  [248] = {x=67.075, y=92.051, z=16.707, rx=-170.912, ry=12.532, rz=153, fatherId=fPrdFrame[0]}
  [249] = {x=69.882, y=92.045, z=17.386, rx=-170.899, ry=12.987, rz=153, fatherId=fPrdFrame[0]}
  [250] = {x=72.688, y=92.04, z=18.091, rx=-170.885, ry=13.443, rz=153, fatherId=fPrdFrame[0]}
  [251] = {x=75.494, y=92.033, z=18.821, rx=-170.871, ry=13.9, rz=153, fatherId=fPrdFrame[0]}
  [252] = {x=78.301, y=92.027, z=19.576, rx=-170.856, ry=14.358, rz=153, fatherId=fPrdFrame[0]}
  [253] = {x=81.107, y=92.021, z=20.356, rx=-170.841, ry=14.816, rz=153, fatherId=fPrdFrame[0]}
  [254] = {x=83.913, y=92.014, z=21.163, rx=-170.825, ry=15.276, rz=153, fatherId=fPrdFrame[0]}
  [255] = {x=86.72, y=92.007, z=21.995, rx=-170.809, ry=15.737, rz=153, fatherId=fPrdFrame[0]}
  [256] = {x=89.526, y=91.999, z=22.854, rx=-170.792, ry=16.198, rz=153, fatherId=fPrdFrame[0]}
  [257] = {x=92.332, y=91.992, z=23.738, rx=-170.774, ry=16.661, rz=153, fatherId=fPrdFrame[0]}
  [258] = {x=95.139, y=91.984, z=24.649, rx=-170.756, ry=17.125, rz=153, fatherId=fPrdFrame[0]}
  [259] = {x=97.945, y=91.976, z=25.587, rx=-170.737, ry=17.59, rz=153, fatherId=fPrdFrame[0]}
  [260] = {x=97.937, y=94.85, z=26.084, rx=-170.445, ry=17.608, rz=153, fatherId=fPrdFrame[0]}
  [261] = {x=95.131, y=94.859, z=25.145, rx=-170.465, ry=17.142, rz=153, fatherId=fPrdFrame[0]}
  [262] = {x=92.325, y=94.867, z=24.233, rx=-170.483, ry=16.678, rz=153, fatherId=fPrdFrame[0]}
  [263] = {x=89.519, y=94.874, z=23.348, rx=-170.501, ry=16.215, rz=153, fatherId=fPrdFrame[0]}
  [264] = {x=86.713, y=94.882, z=22.488, rx=-170.519, ry=15.753, rz=153, fatherId=fPrdFrame[0]}
  [265] = {x=83.907, y=94.889, z=21.655, rx=-170.536, ry=15.292, rz=153, fatherId=fPrdFrame[0]}
  [266] = {x=81.101, y=94.896, z=20.848, rx=-170.552, ry=14.831, rz=153, fatherId=fPrdFrame[0]}
  [267] = {x=78.294, y=94.903, z=20.066, rx=-170.568, ry=14.372, rz=153, fatherId=fPrdFrame[0]}
  [268] = {x=75.488, y=94.909, z=19.31, rx=-170.583, ry=13.914, rz=153, fatherId=fPrdFrame[0]}
  [269] = {x=72.682, y=94.916, z=18.58, rx=-170.598, ry=13.457, rz=153, fatherId=fPrdFrame[0]}
  [270] = {x=69.876, y=94.922, z=17.875, rx=-170.612, ry=13, rz=153, fatherId=fPrdFrame[0]}
  [271] = {x=67.07, y=94.928, z=17.195, rx=-170.625, ry=12.545, rz=153, fatherId=fPrdFrame[0]}
  [272] = {x=64.264, y=94.933, z=16.54, rx=-170.638, ry=12.09, rz=153, fatherId=fPrdFrame[0]}
  [273] = {x=61.458, y=94.939, z=15.909, rx=-170.65, ry=11.636, rz=153, fatherId=fPrdFrame[0]}
  [274] = {x=58.652, y=94.944, z=15.304, rx=-170.662, ry=11.182, rz=153, fatherId=fPrdFrame[0]}
  [275] = {x=55.846, y=94.949, z=14.723, rx=-170.674, ry=10.73, rz=153, fatherId=fPrdFrame[0]}
  [276] = {x=53.04, y=94.953, z=14.167, rx=-170.685, ry=10.278, rz=153, fatherId=fPrdFrame[0]}
  [277] = {x=50.233, y=94.958, z=13.635, rx=-170.695, ry=9.826, rz=153, fatherId=fPrdFrame[0]}
  [278] = {x=47.427, y=94.962, z=13.128, rx=-170.705, ry=9.376, rz=153, fatherId=fPrdFrame[0]}
  [279] = {x=44.621, y=94.966, z=12.645, rx=-170.714, ry=8.925, rz=153, fatherId=fPrdFrame[0]}
  [280] = {x=41.815, y=94.97, z=12.185, rx=-170.723, ry=8.476, rz=153, fatherId=fPrdFrame[0]}
  [281] = {x=39.009, y=94.974, z=11.75, rx=-170.732, ry=8.027, rz=153, fatherId=fPrdFrame[0]}
  [282] = {x=36.203, y=94.977, z=11.339, rx=-170.74, ry=7.578, rz=153, fatherId=fPrdFrame[0]}
  [283] = {x=33.397, y=94.98, z=10.952, rx=-170.747, ry=7.13, rz=153, fatherId=fPrdFrame[0]}
  [284] = {x=30.591, y=94.983, z=10.589, rx=-170.754, ry=6.682, rz=153, fatherId=fPrdFrame[0]}
  [285] = {x=27.785, y=94.986, z=10.249, rx=-170.761, ry=6.235, rz=153, fatherId=fPrdFrame[0]}
  [286] = {x=24.979, y=94.989, z=9.933, rx=-170.767, ry=5.788, rz=153, fatherId=fPrdFrame[0]}
  [287] = {x=22.173, y=94.991, z=9.641, rx=-170.772, ry=5.342, rz=153, fatherId=fPrdFrame[0]}
  [288] = {x=19.367, y=94.993, z=9.372, rx=-170.777, ry=4.895, rz=153, fatherId=fPrdFrame[0]}
  [289] = {x=16.561, y=94.995, z=9.127, rx=-170.782, ry=4.449, rz=153, fatherId=fPrdFrame[0]}
  [290] = {x=13.755, y=94.997, z=8.905, rx=-170.786, ry=4.004, rz=153, fatherId=fPrdFrame[0]}
  [291] = {x=10.948, y=94.999, z=8.707, rx=-170.79, ry=3.558, rz=153, fatherId=fPrdFrame[0]}
  [292] = {x=8.142, y=95, z=8.532, rx=-170.793, ry=3.113, rz=153, fatherId=fPrdFrame[0]}
  [293] = {x=5.336, y=95.001, z=8.381, rx=-170.796, ry=2.668, rz=153, fatherId=fPrdFrame[0]}
  [294] = {x=2.53, y=95.002, z=8.253, rx=-170.799, ry=2.223, rz=153, fatherId=fPrdFrame[0]}
  [295] = {x=-0.276, y=95.003, z=8.148, rx=-170.801, ry=1.778, rz=153, fatherId=fPrdFrame[0]}
  [296] = {x=-3.082, y=95.004, z=8.066, rx=-170.802, ry=1.334, rz=153, fatherId=fPrdFrame[0]}
  [297] = {x=-5.888, y=95.004, z=8.008, rx=-170.803, ry=0.889, rz=153, fatherId=fPrdFrame[0]}
  [298] = {x=-8.694, y=95.005, z=7.973, rx=-170.804, ry=0.444, rz=153, fatherId=fPrdFrame[0]}
  [299] = {x=-11.5, y=95.005, z=7.962, rx=-170.804, rz=153, fatherId=fPrdFrame[0]}
  [300] = {x=-14.306, y=95.005, z=7.973, rx=-170.804, ry=-0.444, rz=153, fatherId=fPrdFrame[0]}
  [301] = {x=-17.112, y=95.004, z=8.008, rx=-170.803, ry=-0.889, rz=153, fatherId=fPrdFrame[0]}
  [302] = {x=-19.918, y=95.004, z=8.066, rx=-170.802, ry=-1.334, rz=153, fatherId=fPrdFrame[0]}
  [303] = {x=-22.724, y=95.003, z=8.148, rx=-170.801, ry=-1.778, rz=153, fatherId=fPrdFrame[0]}
  [304] = {x=-25.53, y=95.002, z=8.253, rx=-170.799, ry=-2.223, rz=153, fatherId=fPrdFrame[0]}
  [305] = {x=-28.336, y=95.001, z=8.381, rx=-170.796, ry=-2.668, rz=153, fatherId=fPrdFrame[0]}
  [306] = {x=-31.142, y=95, z=8.532, rx=-170.793, ry=-3.113, rz=153, fatherId=fPrdFrame[0]}
  [307] = {x=-33.948, y=94.999, z=8.707, rx=-170.79, ry=-3.558, rz=153, fatherId=fPrdFrame[0]}
  [308] = {x=-36.755, y=94.997, z=8.905, rx=-170.786, ry=-4.004, rz=153, fatherId=fPrdFrame[0]}
  [309] = {x=-39.561, y=94.995, z=9.127, rx=-170.782, ry=-4.449, rz=153, fatherId=fPrdFrame[0]}
  [310] = {x=-42.367, y=94.993, z=9.372, rx=-170.777, ry=-4.895, rz=153, fatherId=fPrdFrame[0]}
  [311] = {x=-45.173, y=94.991, z=9.641, rx=-170.772, ry=-5.342, rz=153, fatherId=fPrdFrame[0]}
  [312] = {x=-47.979, y=94.989, z=9.933, rx=-170.767, ry=-5.788, rz=153, fatherId=fPrdFrame[0]}
  [313] = {x=-50.785, y=94.986, z=10.249, rx=-170.761, ry=-6.235, rz=153, fatherId=fPrdFrame[0]}
  [314] = {x=-53.591, y=94.983, z=10.589, rx=-170.754, ry=-6.682, rz=153, fatherId=fPrdFrame[0]}
  [315] = {x=-56.397, y=94.98, z=10.952, rx=-170.747, ry=-7.13, rz=153, fatherId=fPrdFrame[0]}
  [316] = {x=-59.203, y=94.977, z=11.339, rx=-170.74, ry=-7.578, rz=153, fatherId=fPrdFrame[0]}
  [317] = {x=-62.009, y=94.974, z=11.75, rx=-170.732, ry=-8.027, rz=153, fatherId=fPrdFrame[0]}
  [318] = {x=-64.815, y=94.97, z=12.185, rx=-170.723, ry=-8.476, rz=153, fatherId=fPrdFrame[0]}
  [319] = {x=-67.621, y=94.966, z=12.645, rx=-170.714, ry=-8.925, rz=153, fatherId=fPrdFrame[0]}
  [320] = {x=-70.427, y=94.962, z=13.128, rx=-170.705, ry=-9.376, rz=153, fatherId=fPrdFrame[0]}
  [321] = {x=-73.233, y=94.958, z=13.635, rx=-170.695, ry=-9.826, rz=153, fatherId=fPrdFrame[0]}
  [322] = {x=-76.04, y=94.953, z=14.167, rx=-170.685, ry=-10.278, rz=153, fatherId=fPrdFrame[0]}
  [323] = {x=-78.846, y=94.949, z=14.723, rx=-170.674, ry=-10.73, rz=153, fatherId=fPrdFrame[0]}
  [324] = {x=-81.652, y=94.944, z=15.304, rx=-170.662, ry=-11.182, rz=153, fatherId=fPrdFrame[0]}
  [325] = {x=-84.458, y=94.939, z=15.909, rx=-170.65, ry=-11.636, rz=153, fatherId=fPrdFrame[0]}
  [326] = {x=-87.264, y=94.933, z=16.54, rx=-170.638, ry=-12.09, rz=153, fatherId=fPrdFrame[0]}
  [327] = {x=-90.07, y=94.928, z=17.195, rx=-170.625, ry=-12.545, rz=153, fatherId=fPrdFrame[0]}
  [328] = {x=-92.876, y=94.922, z=17.875, rx=-170.612, ry=-13, rz=153, fatherId=fPrdFrame[0]}
  [329] = {x=-95.682, y=94.916, z=18.58, rx=-170.598, ry=-13.457, rz=153, fatherId=fPrdFrame[0]}
  [330] = {x=-98.488, y=94.909, z=19.31, rx=-170.583, ry=-13.914, rz=153, fatherId=fPrdFrame[0]}
  [331] = {x=-101.294, y=94.903, z=20.066, rx=-170.568, ry=-14.372, rz=153, fatherId=fPrdFrame[0]}
  [332] = {x=-104.101, y=94.896, z=20.848, rx=-170.552, ry=-14.831, rz=153, fatherId=fPrdFrame[0]}
  [333] = {x=-106.907, y=94.889, z=21.655, rx=-170.536, ry=-15.292, rz=153, fatherId=fPrdFrame[0]}
  [334] = {x=-109.713, y=94.882, z=22.488, rx=-170.519, ry=-15.753, rz=153, fatherId=fPrdFrame[0]}
  [335] = {x=-112.519, y=94.874, z=23.348, rx=-170.501, ry=-16.215, rz=153, fatherId=fPrdFrame[0]}
  [336] = {x=-115.325, y=94.867, z=24.233, rx=-170.483, ry=-16.678, rz=153, fatherId=fPrdFrame[0]}
  [337] = {x=-118.131, y=94.859, z=25.145, rx=-170.465, ry=-17.142, rz=153, fatherId=fPrdFrame[0]}
  [338] = {x=-120.937, y=94.85, z=26.084, rx=-170.445, ry=-17.608, rz=153, fatherId=fPrdFrame[0]}
  [339] = {x=-120.93, y=97.724, z=26.597, rx=-170.153, ry=-17.627, rz=153, fatherId=fPrdFrame[0]}
  [340] = {x=-118.124, y=97.733, z=25.657, rx=-170.173, ry=-17.161, rz=153, fatherId=fPrdFrame[0]}
  [341] = {x=-115.318, y=97.741, z=24.744, rx=-170.192, ry=-16.696, rz=153, fatherId=fPrdFrame[0]}
  [342] = {x=-112.512, y=97.749, z=23.857, rx=-170.211, ry=-16.232, rz=153, fatherId=fPrdFrame[0]}
  [343] = {x=-109.706, y=97.757, z=22.997, rx=-170.229, ry=-15.769, rz=153, fatherId=fPrdFrame[0]}
  [344] = {x=-106.9, y=97.765, z=22.163, rx=-170.246, ry=-15.308, rz=153, fatherId=fPrdFrame[0]}
  [345] = {x=-104.094, y=97.772, z=21.355, rx=-170.263, ry=-14.847, rz=153, fatherId=fPrdFrame[0]}
  [346] = {x=-101.288, y=97.779, z=20.572, rx=-170.279, ry=-14.387, rz=153, fatherId=fPrdFrame[0]}
  [347] = {x=-98.482, y=97.786, z=19.816, rx=-170.295, ry=-13.929, rz=153, fatherId=fPrdFrame[0]}
  [348] = {x=-95.676, y=97.792, z=19.084, rx=-170.31, ry=-13.471, rz=153, fatherId=fPrdFrame[0]}
  [349] = {x=-92.87, y=97.798, z=18.378, rx=-170.324, ry=-13.014, rz=153, fatherId=fPrdFrame[0]}
  [350] = {x=-90.064, y=97.804, z=17.698, rx=-170.338, ry=-12.558, rz=153, fatherId=fPrdFrame[0]}
  [351] = {x=-87.259, y=97.81, z=17.042, rx=-170.352, ry=-12.102, rz=153, fatherId=fPrdFrame[0]}
  [352] = {x=-84.453, y=97.815, z=16.411, rx=-170.364, ry=-11.648, rz=153, fatherId=fPrdFrame[0]}
  [353] = {x=-81.647, y=97.821, z=15.805, rx=-170.377, ry=-11.194, rz=153, fatherId=fPrdFrame[0]}
  [354] = {x=-78.841, y=97.826, z=15.224, rx=-170.389, ry=-10.741, rz=153, fatherId=fPrdFrame[0]}
  [355] = {x=-76.035, y=97.831, z=14.667, rx=-170.4, ry=-10.288, rz=153, fatherId=fPrdFrame[0]}
  [356] = {x=-73.229, y=97.835, z=14.134, rx=-170.41, ry=-9.837, rz=153, fatherId=fPrdFrame[0]}
  [357] = {x=-70.423, y=97.84, z=13.626, rx=-170.421, ry=-9.385, rz=153, fatherId=fPrdFrame[0]}
  [358] = {x=-67.617, y=97.844, z=13.143, rx=-170.43, ry=-8.935, rz=153, fatherId=fPrdFrame[0]}
  [359] = {x=-64.811, y=97.848, z=12.683, rx=-170.44, ry=-8.485, rz=153, fatherId=fPrdFrame[0]}
  [360] = {x=-62.005, y=97.852, z=12.248, rx=-170.448, ry=-8.035, rz=153, fatherId=fPrdFrame[0]}
  [361] = {x=-59.2, y=97.855, z=11.836, rx=-170.456, ry=-7.586, rz=153, fatherId=fPrdFrame[0]}
  [362] = {x=-56.394, y=97.858, z=11.448, rx=-170.464, ry=-7.137, rz=153, fatherId=fPrdFrame[0]}
  [363] = {x=-53.588, y=97.861, z=11.085, rx=-170.471, ry=-6.689, rz=153, fatherId=fPrdFrame[0]}
  [364] = {x=-50.782, y=97.864, z=10.745, rx=-170.478, ry=-6.242, rz=153, fatherId=fPrdFrame[0]}
  [365] = {x=-47.976, y=97.867, z=10.428, rx=-170.484, ry=-5.794, rz=153, fatherId=fPrdFrame[0]}
  [366] = {x=-45.17, y=97.87, z=10.136, rx=-170.49, ry=-5.347, rz=153, fatherId=fPrdFrame[0]}
  [367] = {x=-42.364, y=97.872, z=9.867, rx=-170.495, ry=-4.9, rz=153, fatherId=fPrdFrame[0]}
  [368] = {x=-39.559, y=97.874, z=9.621, rx=-170.5, ry=-4.454, rz=153, fatherId=fPrdFrame[0]}
  [369] = {x=-36.753, y=97.876, z=9.399, rx=-170.505, ry=-4.008, rz=153, fatherId=fPrdFrame[0]}
  [370] = {x=-33.947, y=97.877, z=9.201, rx=-170.509, ry=-3.562, rz=153, fatherId=fPrdFrame[0]}
  [371] = {x=-31.141, y=97.879, z=9.026, rx=-170.512, ry=-3.116, rz=153, fatherId=fPrdFrame[0]}
  [372] = {x=-28.335, y=97.88, z=8.874, rx=-170.515, ry=-2.671, rz=153, fatherId=fPrdFrame[0]}
  [373] = {x=-25.529, y=97.881, z=8.746, rx=-170.517, ry=-2.225, rz=153, fatherId=fPrdFrame[0]}
  [374] = {x=-22.723, y=97.882, z=8.641, rx=-170.52, ry=-1.78, rz=153, fatherId=fPrdFrame[0]}
  [375] = {x=-19.918, y=97.883, z=8.56, rx=-170.521, ry=-1.335, rz=153, fatherId=fPrdFrame[0]}
  [376] = {x=-17.112, y=97.883, z=8.501, rx=-170.522, ry=-0.89, rz=153, fatherId=fPrdFrame[0]}
  [377] = {x=-14.306, y=97.884, z=8.466, rx=-170.523, ry=-0.445, rz=153, fatherId=fPrdFrame[0]}
  [378] = {x=-11.5, y=97.884, z=8.455, rx=-170.523, rz=153, fatherId=fPrdFrame[0]}
  [379] = {x=-8.694, y=97.884, z=8.466, rx=-170.523, ry=0.445, rz=153, fatherId=fPrdFrame[0]}
  [380] = {x=-5.888, y=97.883, z=8.501, rx=-170.522, ry=0.89, rz=153, fatherId=fPrdFrame[0]}
  [381] = {x=-3.082, y=97.883, z=8.56, rx=-170.521, ry=1.335, rz=153, fatherId=fPrdFrame[0]}
  [382] = {x=-0.277, y=97.882, z=8.641, rx=-170.52, ry=1.78, rz=153, fatherId=fPrdFrame[0]}
  [383] = {x=2.529, y=97.881, z=8.746, rx=-170.517, ry=2.225, rz=153, fatherId=fPrdFrame[0]}
  [384] = {x=5.335, y=97.88, z=8.874, rx=-170.515, ry=2.671, rz=153, fatherId=fPrdFrame[0]}
  [385] = {x=8.141, y=97.879, z=9.026, rx=-170.512, ry=3.116, rz=153, fatherId=fPrdFrame[0]}
  [386] = {x=10.947, y=97.877, z=9.201, rx=-170.509, ry=3.562, rz=153, fatherId=fPrdFrame[0]}
  [387] = {x=13.753, y=97.876, z=9.399, rx=-170.505, ry=4.008, rz=153, fatherId=fPrdFrame[0]}
  [388] = {x=16.559, y=97.874, z=9.621, rx=-170.5, ry=4.454, rz=153, fatherId=fPrdFrame[0]}
  [389] = {x=19.364, y=97.872, z=9.867, rx=-170.495, ry=4.9, rz=153, fatherId=fPrdFrame[0]}
  [390] = {x=22.17, y=97.87, z=10.136, rx=-170.49, ry=5.347, rz=153, fatherId=fPrdFrame[0]}
  [391] = {x=24.976, y=97.867, z=10.428, rx=-170.484, ry=5.794, rz=153, fatherId=fPrdFrame[0]}
  [392] = {x=27.782, y=97.864, z=10.745, rx=-170.478, ry=6.242, rz=153, fatherId=fPrdFrame[0]}
  [393] = {x=30.588, y=97.861, z=11.085, rx=-170.471, ry=6.689, rz=153, fatherId=fPrdFrame[0]}
  [394] = {x=33.394, y=97.858, z=11.448, rx=-170.464, ry=7.137, rz=153, fatherId=fPrdFrame[0]}
  [395] = {x=36.2, y=97.855, z=11.836, rx=-170.456, ry=7.586, rz=153, fatherId=fPrdFrame[0]}
  [396] = {x=39.005, y=97.852, z=12.248, rx=-170.448, ry=8.035, rz=153, fatherId=fPrdFrame[0]}
  [397] = {x=41.811, y=97.848, z=12.683, rx=-170.44, ry=8.485, rz=153, fatherId=fPrdFrame[0]}
  [398] = {x=44.617, y=97.844, z=13.143, rx=-170.43, ry=8.935, rz=153, fatherId=fPrdFrame[0]}
  [399] = {x=47.423, y=97.84, z=13.626, rx=-170.421, ry=9.385, rz=153, fatherId=fPrdFrame[0]}
  [400] = {x=50.229, y=97.835, z=14.134, rx=-170.41, ry=9.837, rz=153, fatherId=fPrdFrame[0]}
  [401] = {x=53.035, y=97.831, z=14.667, rx=-170.4, ry=10.288, rz=153, fatherId=fPrdFrame[0]}
  [402] = {x=55.841, y=97.826, z=15.224, rx=-170.389, ry=10.741, rz=153, fatherId=fPrdFrame[0]}
  [403] = {x=58.647, y=97.821, z=15.805, rx=-170.377, ry=11.194, rz=153, fatherId=fPrdFrame[0]}
  [404] = {x=61.453, y=97.815, z=16.411, rx=-170.364, ry=11.648, rz=153, fatherId=fPrdFrame[0]}
  [405] = {x=64.259, y=97.81, z=17.042, rx=-170.352, ry=12.102, rz=153, fatherId=fPrdFrame[0]}
  [406] = {x=67.064, y=97.804, z=17.698, rx=-170.338, ry=12.558, rz=153, fatherId=fPrdFrame[0]}
  [407] = {x=69.87, y=97.798, z=18.378, rx=-170.324, ry=13.014, rz=153, fatherId=fPrdFrame[0]}
  [408] = {x=72.676, y=97.792, z=19.084, rx=-170.31, ry=13.471, rz=153, fatherId=fPrdFrame[0]}
  [409] = {x=75.482, y=97.786, z=19.816, rx=-170.295, ry=13.929, rz=153, fatherId=fPrdFrame[0]}
  [410] = {x=78.288, y=97.779, z=20.572, rx=-170.279, ry=14.387, rz=153, fatherId=fPrdFrame[0]}
  [411] = {x=81.094, y=97.772, z=21.355, rx=-170.263, ry=14.847, rz=153, fatherId=fPrdFrame[0]}
  [412] = {x=83.9, y=97.765, z=22.163, rx=-170.246, ry=15.308, rz=153, fatherId=fPrdFrame[0]}
  [413] = {x=86.706, y=97.757, z=22.997, rx=-170.229, ry=15.769, rz=153, fatherId=fPrdFrame[0]}
  [414] = {x=89.512, y=97.749, z=23.857, rx=-170.211, ry=16.232, rz=153, fatherId=fPrdFrame[0]}
  [415] = {x=92.318, y=97.741, z=24.744, rx=-170.192, ry=16.696, rz=153, fatherId=fPrdFrame[0]}
  [416] = {x=95.124, y=97.733, z=25.657, rx=-170.173, ry=17.161, rz=153, fatherId=fPrdFrame[0]}
  [417] = {x=97.93, y=97.724, z=26.597, rx=-170.153, ry=17.627, rz=153, fatherId=fPrdFrame[0]}
  [418] = {x=97.922, y=100.599, z=27.126, rx=-169.86, ry=17.646, rz=153, fatherId=fPrdFrame[0]}
  [419] = {x=95.116, y=100.607, z=26.185, rx=-169.881, ry=17.179, rz=153, fatherId=fPrdFrame[0]}
  [420] = {x=92.31, y=100.616, z=25.271, rx=-169.9, ry=16.714, rz=153, fatherId=fPrdFrame[0]}
  [421] = {x=89.504, y=100.624, z=24.383, rx=-169.92, ry=16.25, rz=153, fatherId=fPrdFrame[0]}
  [422] = {x=86.699, y=100.632, z=23.522, rx=-169.938, ry=15.786, rz=153, fatherId=fPrdFrame[0]}
  [423] = {x=83.893, y=100.64, z=22.687, rx=-169.956, ry=15.324, rz=153, fatherId=fPrdFrame[0]}
  [424] = {x=81.087, y=100.647, z=21.877, rx=-169.974, ry=14.863, rz=153, fatherId=fPrdFrame[0]}
  [425] = {x=78.281, y=100.655, z=21.094, rx=-169.99, ry=14.403, rz=153, fatherId=fPrdFrame[0]}
  [426] = {x=75.476, y=100.662, z=20.337, rx=-170.006, ry=13.944, rz=153, fatherId=fPrdFrame[0]}
  [427] = {x=72.67, y=100.668, z=19.604, rx=-170.022, ry=13.485, rz=153, fatherId=fPrdFrame[0]}
  [428] = {x=69.864, y=100.675, z=18.898, rx=-170.037, ry=13.028, rz=153, fatherId=fPrdFrame[0]}
  [429] = {x=67.059, y=100.681, z=18.216, rx=-170.051, ry=12.571, rz=153, fatherId=fPrdFrame[0]}
  [430] = {x=64.253, y=100.687, z=17.56, rx=-170.065, ry=12.116, rz=153, fatherId=fPrdFrame[0]}
  [431] = {x=61.447, y=100.692, z=16.928, rx=-170.078, ry=11.66, rz=153, fatherId=fPrdFrame[0]}
  [432] = {x=58.642, y=100.698, z=16.321, rx=-170.091, ry=11.206, rz=153, fatherId=fPrdFrame[0]}
  [433] = {x=55.836, y=100.703, z=15.739, rx=-170.103, ry=10.752, rz=153, fatherId=fPrdFrame[0]}
  [434] = {x=53.03, y=100.708, z=15.182, rx=-170.115, ry=10.3, rz=153, fatherId=fPrdFrame[0]}
  [435] = {x=50.224, y=100.713, z=14.649, rx=-170.126, ry=9.847, rz=153, fatherId=fPrdFrame[0]}
  [436] = {x=47.419, y=100.717, z=14.14, rx=-170.136, ry=9.396, rz=153, fatherId=fPrdFrame[0]}
  [437] = {x=44.613, y=100.722, z=13.656, rx=-170.146, ry=8.944, rz=153, fatherId=fPrdFrame[0]}
  [438] = {x=41.807, y=100.726, z=13.196, rx=-170.156, ry=8.494, rz=153, fatherId=fPrdFrame[0]}
  [439] = {x=39.002, y=100.73, z=12.76, rx=-170.165, ry=8.044, rz=153, fatherId=fPrdFrame[0]}
  [440] = {x=36.196, y=100.733, z=12.348, rx=-170.173, ry=7.594, rz=153, fatherId=fPrdFrame[0]}
  [441] = {x=33.39, y=100.737, z=11.96, rx=-170.181, ry=7.145, rz=153, fatherId=fPrdFrame[0]}
  [442] = {x=30.585, y=100.74, z=11.596, rx=-170.188, ry=6.696, rz=153, fatherId=fPrdFrame[0]}
  [443] = {x=27.779, y=100.743, z=11.256, rx=-170.195, ry=6.248, rz=153, fatherId=fPrdFrame[0]}
  [444] = {x=24.973, y=100.746, z=10.939, rx=-170.202, ry=5.8, rz=153, fatherId=fPrdFrame[0]}
  [445] = {x=22.168, y=100.748, z=10.646, rx=-170.208, ry=5.353, rz=153, fatherId=fPrdFrame[0]}
  [446] = {x=19.362, y=100.75, z=10.377, rx=-170.213, ry=4.906, rz=153, fatherId=fPrdFrame[0]}
  [447] = {x=16.556, y=100.753, z=10.131, rx=-170.218, ry=4.459, rz=153, fatherId=fPrdFrame[0]}
  [448] = {x=13.751, y=100.754, z=9.909, rx=-170.223, ry=4.012, rz=153, fatherId=fPrdFrame[0]}
  [449] = {x=10.945, y=100.756, z=9.71, rx=-170.227, ry=3.566, rz=153, fatherId=fPrdFrame[0]}
  [450] = {x=8.14, y=100.758, z=9.535, rx=-170.23, ry=3.12, rz=153, fatherId=fPrdFrame[0]}
  [451] = {x=5.334, y=100.759, z=9.383, rx=-170.233, ry=2.674, rz=153, fatherId=fPrdFrame[0]}
  [452] = {x=2.528, y=100.76, z=9.255, rx=-170.236, ry=2.228, rz=153, fatherId=fPrdFrame[0]}
  [453] = {x=-0.277, y=100.761, z=9.15, rx=-170.238, ry=1.782, rz=153, fatherId=fPrdFrame[0]}
  [454] = {x=-3.083, y=100.762, z=9.068, rx=-170.24, ry=1.336, rz=153, fatherId=fPrdFrame[0]}
  [455] = {x=-5.889, y=100.762, z=9.01, rx=-170.241, ry=0.891, rz=153, fatherId=fPrdFrame[0]}
  [456] = {x=-8.694, y=100.763, z=8.975, rx=-170.242, ry=0.445, rz=153, fatherId=fPrdFrame[0]}
  [457] = {x=-11.5, y=100.763, z=8.963, rx=-170.242, rz=153, fatherId=fPrdFrame[0]}
  [458] = {x=-14.306, y=100.763, z=8.975, rx=-170.242, ry=-0.445, rz=153, fatherId=fPrdFrame[0]}
  [459] = {x=-17.111, y=100.762, z=9.01, rx=-170.241, ry=-0.891, rz=153, fatherId=fPrdFrame[0]}
  [460] = {x=-19.917, y=100.762, z=9.068, rx=-170.24, ry=-1.336, rz=153, fatherId=fPrdFrame[0]}
  [461] = {x=-22.723, y=100.761, z=9.15, rx=-170.238, ry=-1.782, rz=153, fatherId=fPrdFrame[0]}
  [462] = {x=-25.528, y=100.76, z=9.255, rx=-170.236, ry=-2.228, rz=153, fatherId=fPrdFrame[0]}
  [463] = {x=-28.334, y=100.759, z=9.383, rx=-170.233, ry=-2.674, rz=153, fatherId=fPrdFrame[0]}
  [464] = {x=-31.14, y=100.758, z=9.535, rx=-170.23, ry=-3.12, rz=153, fatherId=fPrdFrame[0]}
  [465] = {x=-33.945, y=100.756, z=9.71, rx=-170.227, ry=-3.566, rz=153, fatherId=fPrdFrame[0]}
  [466] = {x=-36.751, y=100.754, z=9.909, rx=-170.223, ry=-4.012, rz=153, fatherId=fPrdFrame[0]}
  [467] = {x=-39.556, y=100.753, z=10.131, rx=-170.218, ry=-4.459, rz=153, fatherId=fPrdFrame[0]}
  [468] = {x=-42.362, y=100.75, z=10.377, rx=-170.213, ry=-4.906, rz=153, fatherId=fPrdFrame[0]}
  [469] = {x=-45.168, y=100.748, z=10.646, rx=-170.208, ry=-5.353, rz=153, fatherId=fPrdFrame[0]}
  [470] = {x=-47.973, y=100.746, z=10.939, rx=-170.202, ry=-5.8, rz=153, fatherId=fPrdFrame[0]}
  [471] = {x=-50.779, y=100.743, z=11.256, rx=-170.195, ry=-6.248, rz=153, fatherId=fPrdFrame[0]}
  [472] = {x=-53.585, y=100.74, z=11.596, rx=-170.188, ry=-6.696, rz=153, fatherId=fPrdFrame[0]}
  [473] = {x=-56.39, y=100.737, z=11.96, rx=-170.181, ry=-7.145, rz=153, fatherId=fPrdFrame[0]}
  [474] = {x=-59.196, y=100.733, z=12.348, rx=-170.173, ry=-7.594, rz=153, fatherId=fPrdFrame[0]}
  [475] = {x=-62.002, y=100.73, z=12.76, rx=-170.165, ry=-8.044, rz=153, fatherId=fPrdFrame[0]}
  [476] = {x=-64.807, y=100.726, z=13.196, rx=-170.156, ry=-8.494, rz=153, fatherId=fPrdFrame[0]}
  [477] = {x=-67.613, y=100.722, z=13.656, rx=-170.146, ry=-8.944, rz=153, fatherId=fPrdFrame[0]}
  [478] = {x=-70.419, y=100.717, z=14.14, rx=-170.136, ry=-9.396, rz=153, fatherId=fPrdFrame[0]}
  [479] = {x=-73.224, y=100.713, z=14.649, rx=-170.126, ry=-9.847, rz=153, fatherId=fPrdFrame[0]}
  [480] = {x=-76.03, y=100.708, z=15.182, rx=-170.115, ry=-10.3, rz=153, fatherId=fPrdFrame[0]}
  [481] = {x=-78.836, y=100.703, z=15.739, rx=-170.103, ry=-10.752, rz=153, fatherId=fPrdFrame[0]}
  [482] = {x=-81.642, y=100.698, z=16.321, rx=-170.091, ry=-11.206, rz=153, fatherId=fPrdFrame[0]}
  [483] = {x=-84.447, y=100.692, z=16.928, rx=-170.078, ry=-11.66, rz=153, fatherId=fPrdFrame[0]}
  [484] = {x=-87.253, y=100.687, z=17.56, rx=-170.065, ry=-12.116, rz=153, fatherId=fPrdFrame[0]}
  [485] = {x=-90.059, y=100.681, z=18.216, rx=-170.051, ry=-12.571, rz=153, fatherId=fPrdFrame[0]}
  [486] = {x=-92.864, y=100.675, z=18.898, rx=-170.037, ry=-13.028, rz=153, fatherId=fPrdFrame[0]}
  [487] = {x=-95.67, y=100.668, z=19.604, rx=-170.022, ry=-13.485, rz=153, fatherId=fPrdFrame[0]}
  [488] = {x=-98.476, y=100.662, z=20.337, rx=-170.006, ry=-13.944, rz=153, fatherId=fPrdFrame[0]}
  [489] = {x=-101.281, y=100.655, z=21.094, rx=-169.99, ry=-14.403, rz=153, fatherId=fPrdFrame[0]}
  [490] = {x=-104.087, y=100.647, z=21.877, rx=-169.974, ry=-14.863, rz=153, fatherId=fPrdFrame[0]}
  [491] = {x=-106.893, y=100.64, z=22.687, rx=-169.956, ry=-15.324, rz=153, fatherId=fPrdFrame[0]}
  [492] = {x=-109.699, y=100.632, z=23.522, rx=-169.938, ry=-15.786, rz=153, fatherId=fPrdFrame[0]}
  [493] = {x=-112.504, y=100.624, z=24.383, rx=-169.92, ry=-16.25, rz=153, fatherId=fPrdFrame[0]}
  [494] = {x=-115.31, y=100.616, z=25.271, rx=-169.9, ry=-16.714, rz=153, fatherId=fPrdFrame[0]}
  [495] = {x=-118.116, y=100.607, z=26.185, rx=-169.881, ry=-17.179, rz=153, fatherId=fPrdFrame[0]}
  [496] = {x=-120.922, y=100.599, z=27.126, rx=-169.86, ry=-17.646, rz=153, fatherId=fPrdFrame[0]}
  [497] = {x=-120.922, y=100.599, z=77.126, rx=-169.86, ry=-17.646, rz=153, fatherId=fPrdFrame[0]}
  [498] = {x=19.385, y=66.207, z=5.253, rx=-173.587, ry=4.853, rz=153, fatherId=fPrdFrame[0]}
  [499] = {x=16.577, y=66.209, z=5.01, rx=-173.59, ry=4.411, rz=153, fatherId=fPrdFrame[0]}
  [500] = {x=13.769, y=66.21, z=4.79, rx=-173.593, ry=3.969, rz=153, fatherId=fPrdFrame[0]}
  [501] = {x=10.962, y=66.211, z=4.594, rx=-173.595, ry=3.528, rz=153, fatherId=fPrdFrame[0]}
  [502] = {x=8.154, y=66.212, z=4.42, rx=-173.598, ry=3.086, rz=153, fatherId=fPrdFrame[0]}
  [503] = {x=5.346, y=66.213, z=4.27, rx=-173.6, ry=2.645, rz=153, fatherId=fPrdFrame[0]}
  [504] = {x=2.539, y=66.214, z=4.143, rx=-173.601, ry=2.204, rz=153, fatherId=fPrdFrame[0]}
  [505] = {x=-0.269, y=66.214, z=4.039, rx=-173.603, ry=1.763, rz=153, fatherId=fPrdFrame[0]}
  [506] = {x=-3.077, y=66.215, z=3.958, rx=-173.604, ry=1.322, rz=153, fatherId=fPrdFrame[0]}
  [507] = {x=-5.885, y=66.215, z=3.901, rx=-173.605, ry=0.881, rz=153, fatherId=fPrdFrame[0]}
  [508] = {x=-8.692, y=66.215, z=3.866, rx=-173.605, ry=0.441, rz=153, fatherId=fPrdFrame[0]}
  [509] = {x=-11.5, y=66.215, z=3.855, rx=-173.605, rz=153, fatherId=fPrdFrame[0]}
  [510] = {x=-14.308, y=66.215, z=3.866, rx=-173.605, ry=-0.441, rz=153, fatherId=fPrdFrame[0]}
  [511] = {x=-17.115, y=66.215, z=3.901, rx=-173.605, ry=-0.881, rz=153, fatherId=fPrdFrame[0]}
  [512] = {x=-19.923, y=66.215, z=3.958, rx=-173.604, ry=-1.322, rz=153, fatherId=fPrdFrame[0]}
  [513] = {x=-22.731, y=66.214, z=4.039, rx=-173.603, ry=-1.763, rz=153, fatherId=fPrdFrame[0]}
  [514] = {x=-25.539, y=66.214, z=4.143, rx=-173.601, ry=-2.204, rz=153, fatherId=fPrdFrame[0]}
  [515] = {x=-28.346, y=66.213, z=4.27, rx=-173.6, ry=-2.645, rz=153, fatherId=fPrdFrame[0]}
  [516] = {x=-31.154, y=66.212, z=4.42, rx=-173.598, ry=-3.086, rz=153, fatherId=fPrdFrame[0]}
  [517] = {x=-33.962, y=66.211, z=4.594, rx=-173.595, ry=-3.528, rz=153, fatherId=fPrdFrame[0]}
  [518] = {x=-36.769, y=66.21, z=4.79, rx=-173.593, ry=-3.969, rz=153, fatherId=fPrdFrame[0]}
  [519] = {x=-39.577, y=66.209, z=5.01, rx=-173.59, ry=-4.411, rz=153, fatherId=fPrdFrame[0]}
  [520] = {x=-42.385, y=66.207, z=5.253, rx=-173.587, ry=-4.853, rz=153, fatherId=fPrdFrame[0]}
  [521] = {x=-45.193, y=66.206, z=5.519, rx=-173.583, ry=-5.296, rz=153, fatherId=fPrdFrame[0]}
  [522] = {x=-48, y=66.204, z=5.809, rx=-173.579, ry=-5.738, rz=153, fatherId=fPrdFrame[0]}
  [523] = {x=-50.808, y=66.202, z=6.122, rx=-173.575, ry=-6.181, rz=153, fatherId=fPrdFrame[0]}
  [524] = {x=-53.616, y=66.2, z=6.459, rx=-173.57, ry=-6.625, rz=153, fatherId=fPrdFrame[0]}
  [525] = {x=-56.424, y=66.198, z=6.819, rx=-173.566, ry=-7.069, rz=153, fatherId=fPrdFrame[0]}
  [526] = {x=-59.231, y=66.196, z=7.203, rx=-173.56, ry=-7.513, rz=153, fatherId=fPrdFrame[0]}
  [527] = {x=-62.039, y=66.194, z=7.611, rx=-173.555, ry=-7.958, rz=153, fatherId=fPrdFrame[0]}
  [528] = {x=-64.847, y=66.191, z=8.042, rx=-173.549, ry=-8.403, rz=153, fatherId=fPrdFrame[0]}
  [529] = {x=-67.654, y=66.189, z=8.497, rx=-173.543, ry=-8.848, rz=153, fatherId=fPrdFrame[0]}
  [530] = {x=-70.462, y=66.186, z=8.976, rx=-173.536, ry=-9.295, rz=153, fatherId=fPrdFrame[0]}
  [531] = {x=-73.27, y=66.183, z=9.479, rx=-173.53, ry=-9.742, rz=153, fatherId=fPrdFrame[0]}
  [532] = {x=-76.078, y=66.18, z=10.006, rx=-173.522, ry=-10.189, rz=153, fatherId=fPrdFrame[0]}
  [533] = {x=-78.885, y=66.176, z=10.557, rx=-173.515, ry=-10.637, rz=153, fatherId=fPrdFrame[0]}
  [534] = {x=-81.693, y=66.173, z=11.133, rx=-173.507, ry=-11.086, rz=153, fatherId=fPrdFrame[0]}
  [535] = {x=-84.501, y=66.169, z=11.733, rx=-173.499, ry=-11.535, rz=153, fatherId=fPrdFrame[0]}
  [536] = {x=-87.309, y=66.166, z=12.358, rx=-173.49, ry=-11.985, rz=153, fatherId=fPrdFrame[0]}
  [537] = {x=-90.116, y=66.162, z=13.007, rx=-173.481, ry=-12.436, rz=153, fatherId=fPrdFrame[0]}
  [538] = {x=-92.924, y=66.158, z=13.681, rx=-173.472, ry=-12.887, rz=153, fatherId=fPrdFrame[0]}
  [539] = {x=-95.732, y=66.154, z=14.38, rx=-173.462, ry=-13.34, rz=153, fatherId=fPrdFrame[0]}
  [540] = {x=-98.54, y=66.149, z=15.103, rx=-173.452, ry=-13.793, rz=153, fatherId=fPrdFrame[0]}
  [541] = {x=-101.347, y=66.145, z=15.853, rx=-173.442, ry=-14.247, rz=153, fatherId=fPrdFrame[0]}
  [542] = {x=-104.155, y=66.14, z=16.627, rx=-173.431, ry=-14.702, rz=153, fatherId=fPrdFrame[0]}
  [543] = {x=-106.963, y=66.135, z=17.427, rx=-173.419, ry=-15.158, rz=153, fatherId=fPrdFrame[0]}
  [544] = {x=-109.771, y=66.13, z=18.253, rx=-173.408, ry=-15.615, rz=153, fatherId=fPrdFrame[0]}
  [545] = {x=-112.578, y=66.125, z=19.104, rx=-173.396, ry=-16.073, rz=153, fatherId=fPrdFrame[0]}
  [546] = {x=-115.386, y=66.119, z=19.981, rx=-173.383, ry=-16.532, rz=153, fatherId=fPrdFrame[0]}
  [547] = {x=-118.194, y=66.114, z=20.885, rx=-173.37, ry=-16.992, rz=153, fatherId=fPrdFrame[0]}
  [548] = {x=-121.002, y=66.108, z=21.815, rx=-173.357, ry=-17.454, rz=153, fatherId=fPrdFrame[0]}
  [549] = {x=-120.996, y=68.982, z=22.172, rx=-173.067, ry=-17.466, rz=153, fatherId=fPrdFrame[0]}
  [550] = {x=-118.189, y=68.988, z=21.241, rx=-173.081, ry=-17.005, rz=153, fatherId=fPrdFrame[0]}
  [551] = {x=-115.381, y=68.994, z=20.337, rx=-173.094, ry=-16.544, rz=153, fatherId=fPrdFrame[0]}
  [552] = {x=-112.573, y=69, z=19.459, rx=-173.107, ry=-16.085, rz=153, fatherId=fPrdFrame[0]}
  [553] = {x=-109.766, y=69.005, z=18.607, rx=-173.12, ry=-15.627, rz=153, fatherId=fPrdFrame[0]}
  [554] = {x=-106.958, y=69.01, z=17.781, rx=-173.132, ry=-15.169, rz=153, fatherId=fPrdFrame[0]}
  [555] = {x=-104.151, y=69.016, z=16.98, rx=-173.144, ry=-14.713, rz=153, fatherId=fPrdFrame[0]}
  [556] = {x=-101.343, y=69.02, z=16.205, rx=-173.155, ry=-14.258, rz=153, fatherId=fPrdFrame[0]}
  [557] = {x=-98.535, y=69.025, z=15.455, rx=-173.166, ry=-13.803, rz=153, fatherId=fPrdFrame[0]}
  [558] = {x=-95.728, y=69.03, z=14.731, rx=-173.177, ry=-13.35, rz=153, fatherId=fPrdFrame[0]}
  [559] = {x=-92.92, y=69.034, z=14.032, rx=-173.187, ry=-12.897, rz=153, fatherId=fPrdFrame[0]}
  [560] = {x=-90.112, y=69.038, z=13.357, rx=-173.196, ry=-12.445, rz=153, fatherId=fPrdFrame[0]}
  [561] = {x=-87.305, y=69.042, z=12.707, rx=-173.206, ry=-11.994, rz=153, fatherId=fPrdFrame[0]}
  [562] = {x=-84.497, y=69.046, z=12.082, rx=-173.215, ry=-11.543, rz=153, fatherId=fPrdFrame[0]}
  [563] = {x=-81.69, y=69.05, z=11.482, rx=-173.223, ry=-11.094, rz=153, fatherId=fPrdFrame[0]}
  [564] = {x=-78.882, y=69.054, z=10.906, rx=-173.232, ry=-10.645, rz=153, fatherId=fPrdFrame[0]}
  [565] = {x=-76.074, y=69.057, z=10.354, rx=-173.239, ry=-10.196, rz=153, fatherId=fPrdFrame[0]}
  [566] = {x=-73.267, y=69.06, z=9.827, rx=-173.247, ry=-9.749, rz=153, fatherId=fPrdFrame[0]}
  [567] = {x=-70.459, y=69.063, z=9.323, rx=-173.254, ry=-9.301, rz=153, fatherId=fPrdFrame[0]}
  [568] = {x=-67.652, y=69.066, z=8.844, rx=-173.261, ry=-8.855, rz=153, fatherId=fPrdFrame[0]}
  [569] = {x=-64.844, y=69.069, z=8.389, rx=-173.267, ry=-8.409, rz=153, fatherId=fPrdFrame[0]}
  [570] = {x=-62.037, y=69.072, z=7.957, rx=-173.273, ry=-7.963, rz=153, fatherId=fPrdFrame[0]}
  [571] = {x=-59.229, y=69.074, z=7.549, rx=-173.279, ry=-7.518, rz=153, fatherId=fPrdFrame[0]}
  [572] = {x=-56.421, y=69.077, z=7.165, rx=-173.285, ry=-7.074, rz=153, fatherId=fPrdFrame[0]}
  [573] = {x=-53.614, y=69.079, z=6.805, rx=-173.29, ry=-6.63, rz=153, fatherId=fPrdFrame[0]}
  [574] = {x=-50.806, y=69.081, z=6.468, rx=-173.294, ry=-6.186, rz=153, fatherId=fPrdFrame[0]}
  [575] = {x=-47.999, y=69.083, z=6.154, rx=-173.299, ry=-5.742, rz=153, fatherId=fPrdFrame[0]}
  [576] = {x=-45.191, y=69.084, z=5.864, rx=-173.303, ry=-5.299, rz=153, fatherId=fPrdFrame[0]}
  [577] = {x=-42.383, y=69.086, z=5.598, rx=-173.306, ry=-4.857, rz=153, fatherId=fPrdFrame[0]}
  [578] = {x=-39.576, y=69.087, z=5.354, rx=-173.31, ry=-4.414, rz=153, fatherId=fPrdFrame[0]}
  [579] = {x=-36.768, y=69.089, z=5.135, rx=-173.313, ry=-3.972, rz=153, fatherId=fPrdFrame[0]}
  [580] = {x=-33.961, y=69.09, z=4.938, rx=-173.316, ry=-3.53, rz=153, fatherId=fPrdFrame[0]}
  [581] = {x=-31.153, y=69.091, z=4.764, rx=-173.318, ry=-3.088, rz=153, fatherId=fPrdFrame[0]}
  [582] = {x=-28.345, y=69.092, z=4.614, rx=-173.32, ry=-2.647, rz=153, fatherId=fPrdFrame[0]}
  [583] = {x=-25.538, y=69.093, z=4.487, rx=-173.322, ry=-2.206, rz=153, fatherId=fPrdFrame[0]}
  [584] = {x=-22.73, y=69.093, z=4.383, rx=-173.323, ry=-1.764, rz=153, fatherId=fPrdFrame[0]}
  [585] = {x=-19.923, y=69.094, z=4.302, rx=-173.324, ry=-1.323, rz=153, fatherId=fPrdFrame[0]}
  [586] = {x=-17.115, y=69.094, z=4.244, rx=-173.325, ry=-0.882, rz=153, fatherId=fPrdFrame[0]}
  [587] = {x=-14.308, y=69.094, z=4.21, rx=-173.326, ry=-0.441, rz=153, fatherId=fPrdFrame[0]}
  [588] = {x=-11.5, y=69.094, z=4.198, rx=-173.326, rz=153, fatherId=fPrdFrame[0]}
  [589] = {x=-8.692, y=69.094, z=4.21, rx=-173.326, ry=0.441, rz=153, fatherId=fPrdFrame[0]}
  [590] = {x=-5.885, y=69.094, z=4.244, rx=-173.325, ry=0.882, rz=153, fatherId=fPrdFrame[0]}
  [591] = {x=-3.077, y=69.094, z=4.302, rx=-173.324, ry=1.323, rz=153, fatherId=fPrdFrame[0]}
  [592] = {x=-0.27, y=69.093, z=4.383, rx=-173.323, ry=1.764, rz=153, fatherId=fPrdFrame[0]}
  [593] = {x=2.538, y=69.093, z=4.487, rx=-173.322, ry=2.206, rz=153, fatherId=fPrdFrame[0]}
  [594] = {x=5.345, y=69.092, z=4.614, rx=-173.32, ry=2.647, rz=153, fatherId=fPrdFrame[0]}
  [595] = {x=8.153, y=69.091, z=4.764, rx=-173.318, ry=3.088, rz=153, fatherId=fPrdFrame[0]}
  [596] = {x=10.961, y=69.09, z=4.938, rx=-173.316, ry=3.53, rz=153, fatherId=fPrdFrame[0]}
  [597] = {x=13.768, y=69.089, z=5.135, rx=-173.313, ry=3.972, rz=153, fatherId=fPrdFrame[0]}
  [598] = {x=16.576, y=69.087, z=5.354, rx=-173.31, ry=4.414, rz=153, fatherId=fPrdFrame[0]}
  [599] = {x=19.383, y=69.086, z=5.598, rx=-173.306, ry=4.857, rz=153, fatherId=fPrdFrame[0]}
  [600] = {x=22.191, y=69.084, z=5.864, rx=-173.303, ry=5.299, rz=153, fatherId=fPrdFrame[0]}
  [601] = {x=24.999, y=69.083, z=6.154, rx=-173.299, ry=5.742, rz=153, fatherId=fPrdFrame[0]}
  [602] = {x=27.806, y=69.081, z=6.468, rx=-173.294, ry=6.186, rz=153, fatherId=fPrdFrame[0]}
  [603] = {x=30.614, y=69.079, z=6.805, rx=-173.29, ry=6.63, rz=153, fatherId=fPrdFrame[0]}
  [604] = {x=33.421, y=69.077, z=7.165, rx=-173.285, ry=7.074, rz=153, fatherId=fPrdFrame[0]}
  [605] = {x=36.229, y=69.074, z=7.549, rx=-173.279, ry=7.518, rz=153, fatherId=fPrdFrame[0]}
  [606] = {x=39.037, y=69.072, z=7.957, rx=-173.273, ry=7.963, rz=153, fatherId=fPrdFrame[0]}
  [607] = {x=41.844, y=69.069, z=8.389, rx=-173.267, ry=8.409, rz=153, fatherId=fPrdFrame[0]}
  [608] = {x=44.652, y=69.066, z=8.844, rx=-173.261, ry=8.855, rz=153, fatherId=fPrdFrame[0]}
  [609] = {x=47.459, y=69.063, z=9.323, rx=-173.254, ry=9.301, rz=153, fatherId=fPrdFrame[0]}
  [610] = {x=50.267, y=69.06, z=9.827, rx=-173.247, ry=9.749, rz=153, fatherId=fPrdFrame[0]}
  [611] = {x=53.074, y=69.057, z=10.354, rx=-173.239, ry=10.196, rz=153, fatherId=fPrdFrame[0]}
  [612] = {x=55.882, y=69.054, z=10.906, rx=-173.232, ry=10.645, rz=153, fatherId=fPrdFrame[0]}
  [613] = {x=58.69, y=69.05, z=11.482, rx=-173.223, ry=11.094, rz=153, fatherId=fPrdFrame[0]}
  [614] = {x=61.497, y=69.046, z=12.082, rx=-173.215, ry=11.543, rz=153, fatherId=fPrdFrame[0]}
  [615] = {x=64.305, y=69.042, z=12.707, rx=-173.206, ry=11.994, rz=153, fatherId=fPrdFrame[0]}
  [616] = {x=67.112, y=69.038, z=13.357, rx=-173.196, ry=12.445, rz=153, fatherId=fPrdFrame[0]}
  [617] = {x=69.92, y=69.034, z=14.032, rx=-173.187, ry=12.897, rz=153, fatherId=fPrdFrame[0]}
  [618] = {x=72.728, y=69.03, z=14.731, rx=-173.177, ry=13.35, rz=153, fatherId=fPrdFrame[0]}
  [619] = {x=75.535, y=69.025, z=15.455, rx=-173.166, ry=13.803, rz=153, fatherId=fPrdFrame[0]}
  [620] = {x=78.343, y=69.02, z=16.205, rx=-173.155, ry=14.258, rz=153, fatherId=fPrdFrame[0]}
  [621] = {x=81.151, y=69.016, z=16.98, rx=-173.144, ry=14.713, rz=153, fatherId=fPrdFrame[0]}
  [622] = {x=83.958, y=69.01, z=17.781, rx=-173.132, ry=15.169, rz=153, fatherId=fPrdFrame[0]}
  [623] = {x=86.766, y=69.005, z=18.607, rx=-173.12, ry=15.627, rz=153, fatherId=fPrdFrame[0]}
  [624] = {x=89.573, y=69, z=19.459, rx=-173.107, ry=16.085, rz=153, fatherId=fPrdFrame[0]}
  [625] = {x=92.381, y=68.994, z=20.337, rx=-173.094, ry=16.544, rz=153, fatherId=fPrdFrame[0]}
  [626] = {x=95.189, y=68.988, z=21.241, rx=-173.081, ry=17.005, rz=153, fatherId=fPrdFrame[0]}
  [627] = {x=97.996, y=68.982, z=22.172, rx=-173.067, ry=17.466, rz=153, fatherId=fPrdFrame[0]}
  [628] = {x=97.991, y=71.856, z=22.545, rx=-172.776, ry=17.48, rz=153, fatherId=fPrdFrame[0]}
  [629] = {x=95.183, y=71.863, z=21.613, rx=-172.791, ry=17.018, rz=153, fatherId=fPrdFrame[0]}
  [630] = {x=92.376, y=71.869, z=20.708, rx=-172.805, ry=16.557, rz=153, fatherId=fPrdFrame[0]}
  [631] = {x=89.568, y=71.875, z=19.829, rx=-172.818, ry=16.097, rz=153, fatherId=fPrdFrame[0]}
  [632] = {x=86.761, y=71.88, z=18.977, rx=-172.832, ry=15.639, rz=153, fatherId=fPrdFrame[0]}
  [633] = {x=83.953, y=71.886, z=18.15, rx=-172.844, ry=15.181, rz=153, fatherId=fPrdFrame[0]}
  [634] = {x=81.146, y=71.891, z=17.348, rx=-172.857, ry=14.724, rz=153, fatherId=fPrdFrame[0]}
  [635] = {x=78.338, y=71.896, z=16.573, rx=-172.868, ry=14.268, rz=153, fatherId=fPrdFrame[0]}
  [636] = {x=75.531, y=71.901, z=15.823, rx=-172.88, ry=13.814, rz=153, fatherId=fPrdFrame[0]}
  [637] = {x=72.723, y=71.906, z=15.098, rx=-172.891, ry=13.36, rz=153, fatherId=fPrdFrame[0]}
  [638] = {x=69.916, y=71.911, z=14.398, rx=-172.901, ry=12.907, rz=153, fatherId=fPrdFrame[0]}
  [639] = {x=67.108, y=71.915, z=13.723, rx=-172.912, ry=12.454, rz=153, fatherId=fPrdFrame[0]}
  [640] = {x=64.301, y=71.919, z=13.072, rx=-172.921, ry=12.003, rz=153, fatherId=fPrdFrame[0]}
  [641] = {x=61.494, y=71.923, z=12.447, rx=-172.931, ry=11.552, rz=153, fatherId=fPrdFrame[0]}
  [642] = {x=58.686, y=71.927, z=11.846, rx=-172.94, ry=11.102, rz=153, fatherId=fPrdFrame[0]}
  [643] = {x=55.879, y=71.931, z=11.269, rx=-172.948, ry=10.653, rz=153, fatherId=fPrdFrame[0]}
  [644] = {x=53.071, y=71.934, z=10.717, rx=-172.956, ry=10.204, rz=153, fatherId=fPrdFrame[0]}
  [645] = {x=50.264, y=71.938, z=10.189, rx=-172.964, ry=9.756, rz=153, fatherId=fPrdFrame[0]}
  [646] = {x=47.456, y=71.941, z=9.686, rx=-172.972, ry=9.308, rz=153, fatherId=fPrdFrame[0]}
  [647] = {x=44.649, y=71.944, z=9.206, rx=-172.979, ry=8.862, rz=153, fatherId=fPrdFrame[0]}
  [648] = {x=41.841, y=71.947, z=8.75, rx=-172.985, ry=8.415, rz=153, fatherId=fPrdFrame[0]}
  [649] = {x=39.034, y=71.95, z=8.318, rx=-172.992, ry=7.969, rz=153, fatherId=fPrdFrame[0]}
  [650] = {x=36.226, y=71.952, z=7.91, rx=-172.998, ry=7.524, rz=153, fatherId=fPrdFrame[0]}
  [651] = {x=33.419, y=71.955, z=7.526, rx=-173.003, ry=7.079, rz=153, fatherId=fPrdFrame[0]}
  [652] = {x=30.612, y=71.957, z=7.165, rx=-173.009, ry=6.635, rz=153, fatherId=fPrdFrame[0]}
  [653] = {x=27.804, y=71.959, z=6.828, rx=-173.014, ry=6.191, rz=153, fatherId=fPrdFrame[0]}
  [654] = {x=24.997, y=71.961, z=6.514, rx=-173.018, ry=5.747, rz=153, fatherId=fPrdFrame[0]}
  [655] = {x=22.189, y=71.963, z=6.224, rx=-173.022, ry=5.303, rz=153, fatherId=fPrdFrame[0]}
  [656] = {x=19.382, y=71.965, z=5.957, rx=-173.026, ry=4.86, rz=153, fatherId=fPrdFrame[0]}
  [657] = {x=16.574, y=71.966, z=5.714, rx=-173.03, ry=4.418, rz=153, fatherId=fPrdFrame[0]}
  [658] = {x=13.767, y=71.968, z=5.494, rx=-173.033, ry=3.975, rz=153, fatherId=fPrdFrame[0]}
  [659] = {x=10.959, y=71.969, z=5.297, rx=-173.036, ry=3.533, rz=153, fatherId=fPrdFrame[0]}
  [660] = {x=8.152, y=71.97, z=5.123, rx=-173.038, ry=3.091, rz=153, fatherId=fPrdFrame[0]}
  [661] = {x=5.345, y=71.971, z=4.973, rx=-173.04, ry=2.649, rz=153, fatherId=fPrdFrame[0]}
  [662] = {x=2.537, y=71.972, z=4.846, rx=-173.042, ry=2.207, rz=153, fatherId=fPrdFrame[0]}
  [663] = {x=-0.27, y=71.972, z=4.742, rx=-173.044, ry=1.766, rz=153, fatherId=fPrdFrame[0]}
  [664] = {x=-3.078, y=71.973, z=4.661, rx=-173.045, ry=1.324, rz=153, fatherId=fPrdFrame[0]}
  [665] = {x=-5.885, y=71.973, z=4.603, rx=-173.046, ry=0.883, rz=153, fatherId=fPrdFrame[0]}
  [666] = {x=-8.693, y=71.973, z=4.568, rx=-173.046, ry=0.441, rz=153, fatherId=fPrdFrame[0]}
  [667] = {x=-11.5, y=71.973, z=4.557, rx=-173.046, rz=153, fatherId=fPrdFrame[0]}
  [668] = {x=-14.307, y=71.973, z=4.568, rx=-173.046, ry=-0.441, rz=153, fatherId=fPrdFrame[0]}
  [669] = {x=-17.115, y=71.973, z=4.603, rx=-173.046, ry=-0.883, rz=153, fatherId=fPrdFrame[0]}
  [670] = {x=-19.922, y=71.973, z=4.661, rx=-173.045, ry=-1.324, rz=153, fatherId=fPrdFrame[0]}
  [671] = {x=-22.73, y=71.972, z=4.742, rx=-173.044, ry=-1.766, rz=153, fatherId=fPrdFrame[0]}
  [672] = {x=-25.537, y=71.972, z=4.846, rx=-173.042, ry=-2.207, rz=153, fatherId=fPrdFrame[0]}
  [673] = {x=-28.345, y=71.971, z=4.973, rx=-173.04, ry=-2.649, rz=153, fatherId=fPrdFrame[0]}
  [674] = {x=-31.152, y=71.97, z=5.123, rx=-173.038, ry=-3.091, rz=153, fatherId=fPrdFrame[0]}
  [675] = {x=-33.959, y=71.969, z=5.297, rx=-173.036, ry=-3.533, rz=153, fatherId=fPrdFrame[0]}
  [676] = {x=-36.767, y=71.968, z=5.494, rx=-173.033, ry=-3.975, rz=153, fatherId=fPrdFrame[0]}
  [677] = {x=-39.574, y=71.966, z=5.714, rx=-173.03, ry=-4.418, rz=153, fatherId=fPrdFrame[0]}
  [678] = {x=-42.382, y=71.965, z=5.957, rx=-173.026, ry=-4.86, rz=153, fatherId=fPrdFrame[0]}
  [679] = {x=-45.189, y=71.963, z=6.224, rx=-173.022, ry=-5.303, rz=153, fatherId=fPrdFrame[0]}
  [680] = {x=-47.997, y=71.961, z=6.514, rx=-173.018, ry=-5.747, rz=153, fatherId=fPrdFrame[0]}
  [681] = {x=-50.804, y=71.959, z=6.828, rx=-173.014, ry=-6.191, rz=153, fatherId=fPrdFrame[0]}
  [682] = {x=-53.612, y=71.957, z=7.165, rx=-173.009, ry=-6.635, rz=153, fatherId=fPrdFrame[0]}
  [683] = {x=-56.419, y=71.955, z=7.526, rx=-173.003, ry=-7.079, rz=153, fatherId=fPrdFrame[0]}
  [684] = {x=-59.226, y=71.952, z=7.91, rx=-172.998, ry=-7.524, rz=153, fatherId=fPrdFrame[0]}
  [685] = {x=-62.034, y=71.95, z=8.318, rx=-172.992, ry=-7.969, rz=153, fatherId=fPrdFrame[0]}
  [686] = {x=-64.841, y=71.947, z=8.75, rx=-172.985, ry=-8.415, rz=153, fatherId=fPrdFrame[0]}
  [687] = {x=-67.649, y=71.944, z=9.206, rx=-172.979, ry=-8.862, rz=153, fatherId=fPrdFrame[0]}
  [688] = {x=-70.456, y=71.941, z=9.686, rx=-172.972, ry=-9.308, rz=153, fatherId=fPrdFrame[0]}
  [689] = {x=-73.264, y=71.938, z=10.189, rx=-172.964, ry=-9.756, rz=153, fatherId=fPrdFrame[0]}
  [690] = {x=-76.071, y=71.934, z=10.717, rx=-172.956, ry=-10.204, rz=153, fatherId=fPrdFrame[0]}
  [691] = {x=-78.879, y=71.931, z=11.269, rx=-172.948, ry=-10.653, rz=153, fatherId=fPrdFrame[0]}
  [692] = {x=-81.686, y=71.927, z=11.846, rx=-172.94, ry=-11.102, rz=153, fatherId=fPrdFrame[0]}
  [693] = {x=-84.494, y=71.923, z=12.447, rx=-172.931, ry=-11.552, rz=153, fatherId=fPrdFrame[0]}
  [694] = {x=-87.301, y=71.919, z=13.072, rx=-172.921, ry=-12.003, rz=153, fatherId=fPrdFrame[0]}
  [695] = {x=-90.108, y=71.915, z=13.723, rx=-172.912, ry=-12.454, rz=153, fatherId=fPrdFrame[0]}
  [696] = {x=-92.916, y=71.911, z=14.398, rx=-172.901, ry=-12.907, rz=153, fatherId=fPrdFrame[0]}
  [697] = {x=-95.723, y=71.906, z=15.098, rx=-172.891, ry=-13.36, rz=153, fatherId=fPrdFrame[0]}
  [698] = {x=-98.531, y=71.901, z=15.823, rx=-172.88, ry=-13.814, rz=153, fatherId=fPrdFrame[0]}
  [699] = {x=-101.338, y=71.896, z=16.573, rx=-172.868, ry=-14.268, rz=153, fatherId=fPrdFrame[0]}
  [700] = {x=-104.146, y=71.891, z=17.348, rx=-172.857, ry=-14.724, rz=153, fatherId=fPrdFrame[0]}
  [701] = {x=-106.953, y=71.886, z=18.15, rx=-172.844, ry=-15.181, rz=153, fatherId=fPrdFrame[0]}
  [702] = {x=-109.761, y=71.88, z=18.977, rx=-172.832, ry=-15.639, rz=153, fatherId=fPrdFrame[0]}
  [703] = {x=-112.568, y=71.875, z=19.829, rx=-172.818, ry=-16.097, rz=153, fatherId=fPrdFrame[0]}
  [704] = {x=-115.376, y=71.869, z=20.708, rx=-172.805, ry=-16.557, rz=153, fatherId=fPrdFrame[0]}
  [705] = {x=-118.183, y=71.863, z=21.613, rx=-172.791, ry=-17.018, rz=153, fatherId=fPrdFrame[0]}
  [706] = {x=-120.991, y=71.856, z=22.545, rx=-172.776, ry=-17.48, rz=153, fatherId=fPrdFrame[0]}
  [707] = {x=-120.985, y=74.731, z=22.933, rx=-172.486, ry=-17.494, rz=153, fatherId=fPrdFrame[0]}
  [708] = {x=-118.178, y=74.737, z=22, rx=-172.501, ry=-17.031, rz=153, fatherId=fPrdFrame[0]}
  [709] = {x=-115.37, y=74.744, z=21.095, rx=-172.515, ry=-16.57, rz=153, fatherId=fPrdFrame[0]}
  [710] = {x=-112.563, y=74.75, z=20.215, rx=-172.53, ry=-16.11, rz=153, fatherId=fPrdFrame[0]}
  [711] = {x=-109.756, y=74.756, z=19.362, rx=-172.543, ry=-15.651, rz=153, fatherId=fPrdFrame[0]}
  [712] = {x=-106.948, y=74.761, z=18.534, rx=-172.556, ry=-15.193, rz=153, fatherId=fPrdFrame[0]}
  [713] = {x=-104.141, y=74.767, z=17.732, rx=-172.569, ry=-14.736, rz=153, fatherId=fPrdFrame[0]}
  [714] = {x=-101.334, y=74.772, z=16.956, rx=-172.582, ry=-14.28, rz=153, fatherId=fPrdFrame[0]}
  [715] = {x=-98.526, y=74.777, z=16.205, rx=-172.593, ry=-13.825, rz=153, fatherId=fPrdFrame[0]}
  [716] = {x=-95.719, y=74.782, z=15.479, rx=-172.605, ry=-13.37, rz=153, fatherId=fPrdFrame[0]}
  [717] = {x=-92.912, y=74.787, z=14.779, rx=-172.616, ry=-12.917, rz=153, fatherId=fPrdFrame[0]}
  [718] = {x=-90.104, y=74.792, z=14.103, rx=-172.626, ry=-12.464, rz=153, fatherId=fPrdFrame[0]}
  [719] = {x=-87.297, y=74.796, z=13.452, rx=-172.637, ry=-12.012, rz=153, fatherId=fPrdFrame[0]}
  [720] = {x=-84.49, y=74.8, z=12.826, rx=-172.646, ry=-11.561, rz=153, fatherId=fPrdFrame[0]}
  [721] = {x=-81.682, y=74.804, z=12.225, rx=-172.656, ry=-11.111, rz=153, fatherId=fPrdFrame[0]}
  [722] = {x=-78.875, y=74.808, z=11.648, rx=-172.665, ry=-10.661, rz=153, fatherId=fPrdFrame[0]}
  [723] = {x=-76.068, y=74.812, z=11.096, rx=-172.673, ry=-10.212, rz=153, fatherId=fPrdFrame[0]}
  [724] = {x=-73.26, y=74.815, z=10.567, rx=-172.681, ry=-9.764, rz=153, fatherId=fPrdFrame[0]}
  [725] = {x=-70.453, y=74.819, z=10.063, rx=-172.689, ry=-9.316, rz=153, fatherId=fPrdFrame[0]}
  [726] = {x=-67.646, y=74.822, z=9.583, rx=-172.696, ry=-8.869, rz=153, fatherId=fPrdFrame[0]}
  [727] = {x=-64.839, y=74.825, z=9.127, rx=-172.703, ry=-8.422, rz=153, fatherId=fPrdFrame[0]}
  [728] = {x=-62.031, y=74.828, z=8.695, rx=-172.71, ry=-7.976, rz=153, fatherId=fPrdFrame[0]}
  [729] = {x=-59.224, y=74.83, z=8.286, rx=-172.716, ry=-7.53, rz=153, fatherId=fPrdFrame[0]}
  [730] = {x=-56.417, y=74.833, z=7.901, rx=-172.722, ry=-7.085, rz=153, fatherId=fPrdFrame[0]}
  [731] = {x=-53.609, y=74.835, z=7.54, rx=-172.727, ry=-6.64, rz=153, fatherId=fPrdFrame[0]}
  [732] = {x=-50.802, y=74.837, z=7.203, rx=-172.733, ry=-6.195, rz=153, fatherId=fPrdFrame[0]}
  [733] = {x=-47.995, y=74.84, z=6.889, rx=-172.737, ry=-5.751, rz=153, fatherId=fPrdFrame[0]}
  [734] = {x=-45.187, y=74.841, z=6.599, rx=-172.742, ry=-5.308, rz=153, fatherId=fPrdFrame[0]}
  [735] = {x=-42.38, y=74.843, z=6.332, rx=-172.746, ry=-4.864, rz=153, fatherId=fPrdFrame[0]}
  [736] = {x=-39.573, y=74.845, z=6.088, rx=-172.749, ry=-4.421, rz=153, fatherId=fPrdFrame[0]}
  [737] = {x=-36.766, y=74.846, z=5.868, rx=-172.753, ry=-3.978, rz=153, fatherId=fPrdFrame[0]}
  [738] = {x=-33.958, y=74.847, z=5.671, rx=-172.756, ry=-3.536, rz=153, fatherId=fPrdFrame[0]}
  [739] = {x=-31.151, y=74.849, z=5.497, rx=-172.758, ry=-3.093, rz=153, fatherId=fPrdFrame[0]}
  [740] = {x=-28.344, y=74.85, z=5.347, rx=-172.761, ry=-2.651, rz=153, fatherId=fPrdFrame[0]}
  [741] = {x=-25.536, y=74.85, z=5.219, rx=-172.762, ry=-2.209, rz=153, fatherId=fPrdFrame[0]}
  [742] = {x=-22.729, y=74.851, z=5.115, rx=-172.764, ry=-1.767, rz=153, fatherId=fPrdFrame[0]}
  [743] = {x=-19.922, y=74.852, z=5.034, rx=-172.765, ry=-1.325, rz=153, fatherId=fPrdFrame[0]}
  [744] = {x=-17.115, y=74.852, z=4.976, rx=-172.766, ry=-0.883, rz=153, fatherId=fPrdFrame[0]}
  [745] = {x=-14.307, y=74.852, z=4.942, rx=-172.767, ry=-0.442, rz=153, fatherId=fPrdFrame[0]}
  [746] = {x=-11.5, y=74.852, z=4.93, rx=-172.767, rz=153, fatherId=fPrdFrame[0]}
  [747] = {x=-8.693, y=74.852, z=4.942, rx=-172.767, ry=0.442, rz=153, fatherId=fPrdFrame[0]}
  [748] = {x=-5.885, y=74.852, z=4.976, rx=-172.766, ry=0.883, rz=153, fatherId=fPrdFrame[0]}
  [749] = {x=-3.078, y=74.852, z=5.034, rx=-172.765, ry=1.325, rz=153, fatherId=fPrdFrame[0]}
  [750] = {x=-0.271, y=74.851, z=5.115, rx=-172.764, ry=1.767, rz=153, fatherId=fPrdFrame[0]}
  [751] = {x=2.536, y=74.85, z=5.219, rx=-172.762, ry=2.209, rz=153, fatherId=fPrdFrame[0]}
  [752] = {x=5.344, y=74.85, z=5.347, rx=-172.761, ry=2.651, rz=153, fatherId=fPrdFrame[0]}
  [753] = {x=8.151, y=74.849, z=5.497, rx=-172.758, ry=3.093, rz=153, fatherId=fPrdFrame[0]}
  [754] = {x=10.958, y=74.847, z=5.671, rx=-172.756, ry=3.536, rz=153, fatherId=fPrdFrame[0]}
  [755] = {x=13.766, y=74.846, z=5.868, rx=-172.753, ry=3.978, rz=153, fatherId=fPrdFrame[0]}
  [756] = {x=16.573, y=74.845, z=6.088, rx=-172.749, ry=4.421, rz=153, fatherId=fPrdFrame[0]}
  [757] = {x=19.38, y=74.843, z=6.332, rx=-172.746, ry=4.864, rz=153, fatherId=fPrdFrame[0]}
  [758] = {x=22.187, y=74.841, z=6.599, rx=-172.742, ry=5.308, rz=153, fatherId=fPrdFrame[0]}
  [759] = {x=24.995, y=74.84, z=6.889, rx=-172.737, ry=5.751, rz=153, fatherId=fPrdFrame[0]}
  [760] = {x=27.802, y=74.837, z=7.203, rx=-172.733, ry=6.195, rz=153, fatherId=fPrdFrame[0]}
  [761] = {x=30.609, y=74.835, z=7.54, rx=-172.727, ry=6.64, rz=153, fatherId=fPrdFrame[0]}
  [762] = {x=33.417, y=74.833, z=7.901, rx=-172.722, ry=7.085, rz=153, fatherId=fPrdFrame[0]}
  [763] = {x=36.224, y=74.83, z=8.286, rx=-172.716, ry=7.53, rz=153, fatherId=fPrdFrame[0]}
  [764] = {x=39.031, y=74.828, z=8.695, rx=-172.71, ry=7.976, rz=153, fatherId=fPrdFrame[0]}
  [765] = {x=41.839, y=74.825, z=9.127, rx=-172.703, ry=8.422, rz=153, fatherId=fPrdFrame[0]}
  [766] = {x=44.646, y=74.822, z=9.583, rx=-172.696, ry=8.869, rz=153, fatherId=fPrdFrame[0]}
  [767] = {x=47.453, y=74.819, z=10.063, rx=-172.689, ry=9.316, rz=153, fatherId=fPrdFrame[0]}
  [768] = {x=50.26, y=74.815, z=10.567, rx=-172.681, ry=9.764, rz=153, fatherId=fPrdFrame[0]}
  [769] = {x=53.068, y=74.812, z=11.096, rx=-172.673, ry=10.212, rz=153, fatherId=fPrdFrame[0]}
  [770] = {x=55.875, y=74.808, z=11.648, rx=-172.665, ry=10.661, rz=153, fatherId=fPrdFrame[0]}
  [771] = {x=58.682, y=74.804, z=12.225, rx=-172.656, ry=11.111, rz=153, fatherId=fPrdFrame[0]}
  [772] = {x=61.49, y=74.8, z=12.826, rx=-172.646, ry=11.561, rz=153, fatherId=fPrdFrame[0]}
  [773] = {x=64.297, y=74.796, z=13.452, rx=-172.637, ry=12.012, rz=153, fatherId=fPrdFrame[0]}
  [774] = {x=67.104, y=74.792, z=14.103, rx=-172.626, ry=12.464, rz=153, fatherId=fPrdFrame[0]}
  [775] = {x=69.912, y=74.787, z=14.779, rx=-172.616, ry=12.917, rz=153, fatherId=fPrdFrame[0]}
  [776] = {x=72.719, y=74.782, z=15.479, rx=-172.605, ry=13.37, rz=153, fatherId=fPrdFrame[0]}
  [777] = {x=75.526, y=74.777, z=16.205, rx=-172.593, ry=13.825, rz=153, fatherId=fPrdFrame[0]}
  [778] = {x=78.334, y=74.772, z=16.956, rx=-172.582, ry=14.28, rz=153, fatherId=fPrdFrame[0]}
  [779] = {x=81.141, y=74.767, z=17.732, rx=-172.569, ry=14.736, rz=153, fatherId=fPrdFrame[0]}
  [780] = {x=83.948, y=74.761, z=18.534, rx=-172.556, ry=15.193, rz=153, fatherId=fPrdFrame[0]}
  [781] = {x=86.756, y=74.756, z=19.362, rx=-172.543, ry=15.651, rz=153, fatherId=fPrdFrame[0]}
  [782] = {x=89.563, y=74.75, z=20.215, rx=-172.53, ry=16.11, rz=153, fatherId=fPrdFrame[0]}
  [783] = {x=92.37, y=74.744, z=21.095, rx=-172.515, ry=16.57, rz=153, fatherId=fPrdFrame[0]}
  [784] = {x=95.178, y=74.737, z=22, rx=-172.501, ry=17.031, rz=153, fatherId=fPrdFrame[0]}
  [785] = {x=97.985, y=74.731, z=22.933, rx=-172.486, ry=17.494, rz=153, fatherId=fPrdFrame[0]}
  [786] = {x=97.979, y=77.605, z=23.336, rx=-172.195, ry=17.508, rz=153, fatherId=fPrdFrame[0]}
  [787] = {x=95.172, y=77.612, z=22.403, rx=-172.211, ry=17.046, rz=153, fatherId=fPrdFrame[0]}
  [788] = {x=92.364, y=77.618, z=21.496, rx=-172.226, ry=16.584, rz=153, fatherId=fPrdFrame[0]}
  [789] = {x=89.557, y=77.625, z=20.616, rx=-172.24, ry=16.123, rz=153, fatherId=fPrdFrame[0]}
  [790] = {x=86.75, y=77.631, z=19.762, rx=-172.255, ry=15.664, rz=153, fatherId=fPrdFrame[0]}
  [791] = {x=83.943, y=77.637, z=18.934, rx=-172.268, ry=15.206, rz=153, fatherId=fPrdFrame[0]}
  [792] = {x=81.136, y=77.642, z=18.131, rx=-172.282, ry=14.748, rz=153, fatherId=fPrdFrame[0]}
  [793] = {x=78.329, y=77.648, z=17.354, rx=-172.295, ry=14.292, rz=153, fatherId=fPrdFrame[0]}
  [794] = {x=75.521, y=77.653, z=16.603, rx=-172.307, ry=13.836, rz=153, fatherId=fPrdFrame[0]}
  [795] = {x=72.714, y=77.658, z=15.876, rx=-172.319, ry=13.381, rz=153, fatherId=fPrdFrame[0]}
  [796] = {x=69.907, y=77.663, z=15.175, rx=-172.33, ry=12.927, rz=153, fatherId=fPrdFrame[0]}
  [797] = {x=67.1, y=77.668, z=14.499, rx=-172.341, ry=12.474, rz=153, fatherId=fPrdFrame[0]}
  [798] = {x=64.293, y=77.673, z=13.848, rx=-172.352, ry=12.022, rz=153, fatherId=fPrdFrame[0]}
  [799] = {x=61.486, y=77.677, z=13.221, rx=-172.362, ry=11.571, rz=153, fatherId=fPrdFrame[0]}
  [800] = {x=58.678, y=77.681, z=12.619, rx=-172.372, ry=11.12, rz=153, fatherId=fPrdFrame[0]}
  [801] = {x=55.871, y=77.685, z=12.042, rx=-172.381, ry=10.67, rz=153, fatherId=fPrdFrame[0]}
  [802] = {x=53.064, y=77.689, z=11.489, rx=-172.39, ry=10.22, rz=153, fatherId=fPrdFrame[0]}
  [803] = {x=50.257, y=77.693, z=10.96, rx=-172.398, ry=9.772, rz=153, fatherId=fPrdFrame[0]}
  [804] = {x=47.45, y=77.696, z=10.455, rx=-172.406, ry=9.323, rz=153, fatherId=fPrdFrame[0]}
  [805] = {x=44.643, y=77.7, z=9.975, rx=-172.414, ry=8.876, rz=153, fatherId=fPrdFrame[0]}
  [806] = {x=41.836, y=77.703, z=9.518, rx=-172.421, ry=8.429, rz=153, fatherId=fPrdFrame[0]}
  [807] = {x=39.028, y=77.706, z=9.086, rx=-172.428, ry=7.982, rz=153, fatherId=fPrdFrame[0]}
  [808] = {x=36.221, y=77.708, z=8.677, rx=-172.434, ry=7.536, rz=153, fatherId=fPrdFrame[0]}
  [809] = {x=33.414, y=77.711, z=8.292, rx=-172.44, ry=7.09, rz=153, fatherId=fPrdFrame[0]}
  [810] = {x=30.607, y=77.714, z=7.931, rx=-172.446, ry=6.645, rz=153, fatherId=fPrdFrame[0]}
  [811] = {x=27.8, y=77.716, z=7.593, rx=-172.451, ry=6.2, rz=153, fatherId=fPrdFrame[0]}
  [812] = {x=24.993, y=77.718, z=7.279, rx=-172.456, ry=5.756, rz=153, fatherId=fPrdFrame[0]}
  [813] = {x=22.186, y=77.72, z=6.988, rx=-172.461, ry=5.312, rz=153, fatherId=fPrdFrame[0]}
  [814] = {x=19.378, y=77.722, z=6.721, rx=-172.465, ry=4.868, rz=153, fatherId=fPrdFrame[0]}
  [815] = {x=16.571, y=77.723, z=6.477, rx=-172.469, ry=4.425, rz=153, fatherId=fPrdFrame[0]}
  [816] = {x=13.764, y=77.725, z=6.257, rx=-172.472, ry=3.981, rz=153, fatherId=fPrdFrame[0]}
  [817] = {x=10.957, y=77.726, z=6.06, rx=-172.475, ry=3.538, rz=153, fatherId=fPrdFrame[0]}
  [818] = {x=8.15, y=77.727, z=5.886, rx=-172.478, ry=3.096, rz=153, fatherId=fPrdFrame[0]}
  [819] = {x=5.343, y=77.728, z=5.735, rx=-172.481, ry=2.653, rz=153, fatherId=fPrdFrame[0]}
  [820] = {x=2.536, y=77.729, z=5.608, rx=-172.483, ry=2.211, rz=153, fatherId=fPrdFrame[0]}
  [821] = {x=-0.271, y=77.73, z=5.503, rx=-172.484, ry=1.768, rz=153, fatherId=fPrdFrame[0]}
  [822] = {x=-3.079, y=77.731, z=5.422, rx=-172.485, ry=1.326, rz=153, fatherId=fPrdFrame[0]}
  [823] = {x=-5.886, y=77.731, z=5.365, rx=-172.486, ry=0.884, rz=153, fatherId=fPrdFrame[0]}
  [824] = {x=-8.693, y=77.731, z=5.33, rx=-172.487, ry=0.442, rz=153, fatherId=fPrdFrame[0]}
  [825] = {x=-11.5, y=77.731, z=5.318, rx=-172.487, rz=153, fatherId=fPrdFrame[0]}
  [826] = {x=-14.307, y=77.731, z=5.33, rx=-172.487, ry=-0.442, rz=153, fatherId=fPrdFrame[0]}
  [827] = {x=-17.114, y=77.731, z=5.365, rx=-172.486, ry=-0.884, rz=153, fatherId=fPrdFrame[0]}
  [828] = {x=-19.921, y=77.731, z=5.422, rx=-172.485, ry=-1.326, rz=153, fatherId=fPrdFrame[0]}
  [829] = {x=-22.729, y=77.73, z=5.503, rx=-172.484, ry=-1.768, rz=153, fatherId=fPrdFrame[0]}
  [830] = {x=-25.536, y=77.729, z=5.608, rx=-172.483, ry=-2.211, rz=153, fatherId=fPrdFrame[0]}
  [831] = {x=-28.343, y=77.728, z=5.735, rx=-172.481, ry=-2.653, rz=153, fatherId=fPrdFrame[0]}
  [832] = {x=-31.15, y=77.727, z=5.886, rx=-172.478, ry=-3.096, rz=153, fatherId=fPrdFrame[0]}
  [833] = {x=-33.957, y=77.726, z=6.06, rx=-172.475, ry=-3.538, rz=153, fatherId=fPrdFrame[0]}
  [834] = {x=-36.764, y=77.725, z=6.257, rx=-172.472, ry=-3.981, rz=153, fatherId=fPrdFrame[0]}
  [835] = {x=-39.571, y=77.723, z=6.477, rx=-172.469, ry=-4.425, rz=153, fatherId=fPrdFrame[0]}
  [836] = {x=-42.378, y=77.722, z=6.721, rx=-172.465, ry=-4.868, rz=153, fatherId=fPrdFrame[0]}
  [837] = {x=-45.186, y=77.72, z=6.988, rx=-172.461, ry=-5.312, rz=153, fatherId=fPrdFrame[0]}
  [838] = {x=-47.993, y=77.718, z=7.279, rx=-172.456, ry=-5.756, rz=153, fatherId=fPrdFrame[0]}
  [839] = {x=-50.8, y=77.716, z=7.593, rx=-172.451, ry=-6.2, rz=153, fatherId=fPrdFrame[0]}
  [840] = {x=-53.607, y=77.714, z=7.931, rx=-172.446, ry=-6.645, rz=153, fatherId=fPrdFrame[0]}
  [841] = {x=-56.414, y=77.711, z=8.292, rx=-172.44, ry=-7.09, rz=153, fatherId=fPrdFrame[0]}
  [842] = {x=-59.221, y=77.708, z=8.677, rx=-172.434, ry=-7.536, rz=153, fatherId=fPrdFrame[0]}
  [843] = {x=-62.028, y=77.706, z=9.086, rx=-172.428, ry=-7.982, rz=153, fatherId=fPrdFrame[0]}
  [844] = {x=-64.836, y=77.703, z=9.518, rx=-172.421, ry=-8.429, rz=153, fatherId=fPrdFrame[0]}
  [845] = {x=-67.643, y=77.7, z=9.975, rx=-172.414, ry=-8.876, rz=153, fatherId=fPrdFrame[0]}
  [846] = {x=-70.45, y=77.696, z=10.455, rx=-172.406, ry=-9.323, rz=153, fatherId=fPrdFrame[0]}
  [847] = {x=-73.257, y=77.693, z=10.96, rx=-172.398, ry=-9.772, rz=153, fatherId=fPrdFrame[0]}
  [848] = {x=-76.064, y=77.689, z=11.489, rx=-172.39, ry=-10.22, rz=153, fatherId=fPrdFrame[0]}
  [849] = {x=-78.871, y=77.685, z=12.042, rx=-172.381, ry=-10.67, rz=153, fatherId=fPrdFrame[0]}
  [850] = {x=-81.678, y=77.681, z=12.619, rx=-172.372, ry=-11.12, rz=153, fatherId=fPrdFrame[0]}
  [851] = {x=-84.486, y=77.677, z=13.221, rx=-172.362, ry=-11.571, rz=153, fatherId=fPrdFrame[0]}
  [852] = {x=-87.293, y=77.673, z=13.848, rx=-172.352, ry=-12.022, rz=153, fatherId=fPrdFrame[0]}
  [853] = {x=-90.1, y=77.668, z=14.499, rx=-172.341, ry=-12.474, rz=153, fatherId=fPrdFrame[0]}
  [854] = {x=-92.907, y=77.663, z=15.175, rx=-172.33, ry=-12.927, rz=153, fatherId=fPrdFrame[0]}
  [855] = {x=-95.714, y=77.658, z=15.876, rx=-172.319, ry=-13.381, rz=153, fatherId=fPrdFrame[0]}
  [856] = {x=-98.521, y=77.653, z=16.603, rx=-172.307, ry=-13.836, rz=153, fatherId=fPrdFrame[0]}
  [857] = {x=-101.329, y=77.648, z=17.354, rx=-172.295, ry=-14.292, rz=153, fatherId=fPrdFrame[0]}
  [858] = {x=-104.136, y=77.642, z=18.131, rx=-172.282, ry=-14.748, rz=153, fatherId=fPrdFrame[0]}
  [859] = {x=-106.943, y=77.637, z=18.934, rx=-172.268, ry=-15.206, rz=153, fatherId=fPrdFrame[0]}
  [860] = {x=-109.75, y=77.631, z=19.762, rx=-172.255, ry=-15.664, rz=153, fatherId=fPrdFrame[0]}
  [861] = {x=-112.557, y=77.625, z=20.616, rx=-172.24, ry=-16.123, rz=153, fatherId=fPrdFrame[0]}
  [862] = {x=-115.364, y=77.618, z=21.496, rx=-172.226, ry=-16.584, rz=153, fatherId=fPrdFrame[0]}
  [863] = {x=-118.172, y=77.612, z=22.403, rx=-172.211, ry=-17.046, rz=153, fatherId=fPrdFrame[0]}
  [864] = {x=-120.979, y=77.605, z=23.336, rx=-172.195, ry=-17.508, rz=153, fatherId=fPrdFrame[0]}
  [865] = {x=-120.973, y=80.479, z=23.755, rx=-171.904, ry=-17.523, rz=153, fatherId=fPrdFrame[0]}
  [866] = {x=-118.166, y=80.486, z=22.821, rx=-171.92, ry=-17.06, rz=153, fatherId=fPrdFrame[0]}
  [867] = {x=-115.359, y=80.493, z=21.914, rx=-171.936, ry=-16.598, rz=153, fatherId=fPrdFrame[0]}
  [868] = {x=-112.551, y=80.5, z=21.033, rx=-171.951, ry=-16.137, rz=153, fatherId=fPrdFrame[0]}
  [869] = {x=-109.744, y=80.506, z=20.178, rx=-171.966, ry=-15.677, rz=153, fatherId=fPrdFrame[0]}
  [870] = {x=-106.937, y=80.512, z=19.349, rx=-171.98, ry=-15.219, rz=153, fatherId=fPrdFrame[0]}
  [871] = {x=-104.13, y=80.518, z=18.545, rx=-171.994, ry=-14.761, rz=153, fatherId=fPrdFrame[0]}
  [872] = {x=-101.323, y=80.524, z=17.768, rx=-172.007, ry=-14.304, rz=153, fatherId=fPrdFrame[0]}
  [873] = {x=-98.516, y=80.529, z=17.015, rx=-172.02, ry=-13.848, rz=153, fatherId=fPrdFrame[0]}
  [874] = {x=-95.709, y=80.535, z=16.289, rx=-172.032, ry=-13.393, rz=153, fatherId=fPrdFrame[0]}
  [875] = {x=-92.902, y=80.54, z=15.587, rx=-172.044, ry=-12.938, rz=153, fatherId=fPrdFrame[0]}
  [876] = {x=-90.095, y=80.545, z=14.91, rx=-172.056, ry=-12.485, rz=153, fatherId=fPrdFrame[0]}
  [877] = {x=-87.288, y=80.549, z=14.258, rx=-172.067, ry=-12.032, rz=153, fatherId=fPrdFrame[0]}
  [878] = {x=-84.481, y=80.554, z=13.631, rx=-172.077, ry=-11.581, rz=153, fatherId=fPrdFrame[0]}
  [879] = {x=-81.674, y=80.558, z=13.029, rx=-172.087, ry=-11.129, rz=153, fatherId=fPrdFrame[0]}
  [880] = {x=-78.867, y=80.563, z=12.451, rx=-172.097, ry=-10.679, rz=153, fatherId=fPrdFrame[0]}
  [881] = {x=-76.06, y=80.566, z=11.897, rx=-172.106, ry=-10.229, rz=153, fatherId=fPrdFrame[0]}
  [882] = {x=-73.253, y=80.57, z=11.368, rx=-172.115, ry=-9.78, rz=153, fatherId=fPrdFrame[0]}
  [883] = {x=-70.446, y=80.574, z=10.863, rx=-172.123, ry=-9.331, rz=153, fatherId=fPrdFrame[0]}
  [884] = {x=-67.639, y=80.577, z=10.382, rx=-172.131, ry=-8.883, rz=153, fatherId=fPrdFrame[0]}
  [885] = {x=-64.832, y=80.581, z=9.925, rx=-172.139, ry=-8.436, rz=153, fatherId=fPrdFrame[0]}
  [886] = {x=-62.025, y=80.584, z=9.492, rx=-172.146, ry=-7.989, rz=153, fatherId=fPrdFrame[0]}
  [887] = {x=-59.218, y=80.587, z=9.083, rx=-172.152, ry=-7.542, rz=153, fatherId=fPrdFrame[0]}
  [888] = {x=-56.412, y=80.589, z=8.698, rx=-172.159, ry=-7.096, rz=153, fatherId=fPrdFrame[0]}
  [889] = {x=-53.605, y=80.592, z=8.336, rx=-172.165, ry=-6.651, rz=153, fatherId=fPrdFrame[0]}
  [890] = {x=-50.798, y=80.594, z=7.998, rx=-172.17, ry=-6.206, rz=153, fatherId=fPrdFrame[0]}
  [891] = {x=-47.991, y=80.596, z=7.684, rx=-172.175, ry=-5.761, rz=153, fatherId=fPrdFrame[0]}
  [892] = {x=-45.184, y=80.598, z=7.393, rx=-172.18, ry=-5.316, rz=153, fatherId=fPrdFrame[0]}
  [893] = {x=-42.377, y=80.6, z=7.125, rx=-172.184, ry=-4.872, rz=153, fatherId=fPrdFrame[0]}
  [894] = {x=-39.57, y=80.602, z=6.881, rx=-172.188, ry=-4.428, rz=153, fatherId=fPrdFrame[0]}
  [895] = {x=-36.763, y=80.604, z=6.661, rx=-172.192, ry=-3.985, rz=153, fatherId=fPrdFrame[0]}
  [896] = {x=-33.956, y=80.605, z=6.463, rx=-172.195, ry=-3.541, rz=153, fatherId=fPrdFrame[0]}
  [897] = {x=-31.149, y=80.606, z=6.289, rx=-172.198, ry=-3.098, rz=153, fatherId=fPrdFrame[0]}
  [898] = {x=-28.342, y=80.607, z=6.139, rx=-172.2, ry=-2.655, rz=153, fatherId=fPrdFrame[0]}
  [899] = {x=-25.535, y=80.608, z=6.011, rx=-172.202, ry=-2.213, rz=153, fatherId=fPrdFrame[0]}
  [900] = {x=-22.728, y=80.609, z=5.907, rx=-172.204, ry=-1.77, rz=153, fatherId=fPrdFrame[0]}
  [901] = {x=-19.921, y=80.609, z=5.826, rx=-172.205, ry=-1.327, rz=153, fatherId=fPrdFrame[0]}
  [902] = {x=-17.114, y=80.61, z=5.768, rx=-172.206, ry=-0.885, rz=153, fatherId=fPrdFrame[0]}
  [903] = {x=-14.307, y=80.61, z=5.733, rx=-172.207, ry=-0.442, rz=153, fatherId=fPrdFrame[0]}
  [904] = {x=-11.5, y=80.61, z=5.721, rx=-172.207, rz=153, fatherId=fPrdFrame[0]}
  [905] = {x=-8.693, y=80.61, z=5.733, rx=-172.207, ry=0.442, rz=153, fatherId=fPrdFrame[0]}
  [906] = {x=-5.886, y=80.61, z=5.768, rx=-172.206, ry=0.885, rz=153, fatherId=fPrdFrame[0]}
  [907] = {x=-3.079, y=80.609, z=5.826, rx=-172.205, ry=1.327, rz=153, fatherId=fPrdFrame[0]}
  [908] = {x=-0.272, y=80.609, z=5.907, rx=-172.204, ry=1.77, rz=153, fatherId=fPrdFrame[0]}
  [909] = {x=2.535, y=80.608, z=6.011, rx=-172.202, ry=2.213, rz=153, fatherId=fPrdFrame[0]}
  [910] = {x=5.342, y=80.607, z=6.139, rx=-172.2, ry=2.655, rz=153, fatherId=fPrdFrame[0]}
  [911] = {x=8.149, y=80.606, z=6.289, rx=-172.198, ry=3.098, rz=153, fatherId=fPrdFrame[0]}
  [912] = {x=10.956, y=80.605, z=6.463, rx=-172.195, ry=3.541, rz=153, fatherId=fPrdFrame[0]}
  [913] = {x=13.763, y=80.604, z=6.661, rx=-172.192, ry=3.985, rz=153, fatherId=fPrdFrame[0]}
  [914] = {x=16.57, y=80.602, z=6.881, rx=-172.188, ry=4.428, rz=153, fatherId=fPrdFrame[0]}
  [915] = {x=19.377, y=80.6, z=7.125, rx=-172.184, ry=4.872, rz=153, fatherId=fPrdFrame[0]}
  [916] = {x=22.184, y=80.598, z=7.393, rx=-172.18, ry=5.316, rz=153, fatherId=fPrdFrame[0]}
  [917] = {x=24.991, y=80.596, z=7.684, rx=-172.175, ry=5.761, rz=153, fatherId=fPrdFrame[0]}
  [918] = {x=27.798, y=80.594, z=7.998, rx=-172.17, ry=6.206, rz=153, fatherId=fPrdFrame[0]}
  [919] = {x=30.605, y=80.592, z=8.336, rx=-172.165, ry=6.651, rz=153, fatherId=fPrdFrame[0]}
  [920] = {x=33.412, y=80.589, z=8.698, rx=-172.159, ry=7.096, rz=153, fatherId=fPrdFrame[0]}
  [921] = {x=36.218, y=80.587, z=9.083, rx=-172.152, ry=7.542, rz=153, fatherId=fPrdFrame[0]}
  [922] = {x=39.025, y=80.584, z=9.492, rx=-172.146, ry=7.989, rz=153, fatherId=fPrdFrame[0]}
  [923] = {x=41.832, y=80.581, z=9.925, rx=-172.139, ry=8.436, rz=153, fatherId=fPrdFrame[0]}
  [924] = {x=44.639, y=80.577, z=10.382, rx=-172.131, ry=8.883, rz=153, fatherId=fPrdFrame[0]}
  [925] = {x=47.446, y=80.574, z=10.863, rx=-172.123, ry=9.331, rz=153, fatherId=fPrdFrame[0]}
  [926] = {x=50.253, y=80.57, z=11.368, rx=-172.115, ry=9.78, rz=153, fatherId=fPrdFrame[0]}
  [927] = {x=53.06, y=80.566, z=11.897, rx=-172.106, ry=10.229, rz=153, fatherId=fPrdFrame[0]}
  [928] = {x=55.867, y=80.563, z=12.451, rx=-172.097, ry=10.679, rz=153, fatherId=fPrdFrame[0]}
  [929] = {x=58.674, y=80.558, z=13.029, rx=-172.087, ry=11.129, rz=153, fatherId=fPrdFrame[0]}
  [930] = {x=61.481, y=80.554, z=13.631, rx=-172.077, ry=11.581, rz=153, fatherId=fPrdFrame[0]}
  [931] = {x=64.288, y=80.549, z=14.258, rx=-172.067, ry=12.032, rz=153, fatherId=fPrdFrame[0]}
  [932] = {x=67.095, y=80.545, z=14.91, rx=-172.056, ry=12.485, rz=153, fatherId=fPrdFrame[0]}
  [933] = {x=69.902, y=80.54, z=15.587, rx=-172.044, ry=12.938, rz=153, fatherId=fPrdFrame[0]}
  [934] = {x=72.709, y=80.535, z=16.289, rx=-172.032, ry=13.393, rz=153, fatherId=fPrdFrame[0]}
  [935] = {x=75.516, y=80.529, z=17.015, rx=-172.02, ry=13.848, rz=153, fatherId=fPrdFrame[0]}
  [936] = {x=78.323, y=80.524, z=17.768, rx=-172.007, ry=14.304, rz=153, fatherId=fPrdFrame[0]}
  [937] = {x=81.13, y=80.518, z=18.545, rx=-171.994, ry=14.761, rz=153, fatherId=fPrdFrame[0]}
  [938] = {x=83.937, y=80.512, z=19.349, rx=-171.98, ry=15.219, rz=153, fatherId=fPrdFrame[0]}
  [939] = {x=86.744, y=80.506, z=20.178, rx=-171.966, ry=15.677, rz=153, fatherId=fPrdFrame[0]}
  [940] = {x=89.551, y=80.5, z=21.033, rx=-171.951, ry=16.137, rz=153, fatherId=fPrdFrame[0]}
  [941] = {x=92.359, y=80.493, z=21.914, rx=-171.936, ry=16.598, rz=153, fatherId=fPrdFrame[0]}
  [942] = {x=95.166, y=80.486, z=22.821, rx=-171.92, ry=17.06, rz=153, fatherId=fPrdFrame[0]}
  [943] = {x=97.973, y=80.479, z=23.755, rx=-171.904, ry=17.523, rz=153, fatherId=fPrdFrame[0]}
  [944] = {x=97.966, y=83.353, z=24.19, rx=-171.612, ry=17.539, rz=153, fatherId=fPrdFrame[0]}
  [945] = {x=95.159, y=83.361, z=23.255, rx=-171.629, ry=17.076, rz=153, fatherId=fPrdFrame[0]}
  [946] = {x=92.352, y=83.368, z=22.346, rx=-171.646, ry=16.613, rz=153, fatherId=fPrdFrame[0]}
  [947] = {x=89.545, y=83.375, z=21.465, rx=-171.662, ry=16.152, rz=153, fatherId=fPrdFrame[0]}
  [948] = {x=86.739, y=83.381, z=20.609, rx=-171.677, ry=15.691, rz=153, fatherId=fPrdFrame[0]}
  [949] = {x=83.932, y=83.388, z=19.779, rx=-171.692, ry=15.232, rz=153, fatherId=fPrdFrame[0]}
  [950] = {x=81.125, y=83.394, z=18.975, rx=-171.706, ry=14.774, rz=153, fatherId=fPrdFrame[0]}
  [951] = {x=78.318, y=83.4, z=18.197, rx=-171.72, ry=14.317, rz=153, fatherId=fPrdFrame[0]}
  [952] = {x=75.511, y=83.405, z=17.444, rx=-171.733, ry=13.86, rz=153, fatherId=fPrdFrame[0]}
  [953] = {x=72.704, y=83.411, z=16.716, rx=-171.746, ry=13.405, rz=153, fatherId=fPrdFrame[0]}
  [954] = {x=69.897, y=83.416, z=16.014, rx=-171.758, ry=12.95, rz=153, fatherId=fPrdFrame[0]}
  [955] = {x=67.091, y=83.421, z=15.336, rx=-171.77, ry=12.496, rz=153, fatherId=fPrdFrame[0]}
  [956] = {x=64.284, y=83.426, z=14.684, rx=-171.781, ry=12.043, rz=153, fatherId=fPrdFrame[0]}
  [957] = {x=61.477, y=83.431, z=14.056, rx=-171.792, ry=11.591, rz=153, fatherId=fPrdFrame[0]}
  [958] = {x=58.67, y=83.435, z=13.453, rx=-171.803, ry=11.139, rz=153, fatherId=fPrdFrame[0]}
  [959] = {x=55.863, y=83.44, z=12.875, rx=-171.813, ry=10.688, rz=153, fatherId=fPrdFrame[0]}
  [960] = {x=53.057, y=83.444, z=12.321, rx=-171.822, ry=10.238, rz=153, fatherId=fPrdFrame[0]}
  [961] = {x=50.25, y=83.448, z=11.791, rx=-171.831, ry=9.789, rz=153, fatherId=fPrdFrame[0]}
  [962] = {x=47.443, y=83.452, z=11.286, rx=-171.84, ry=9.34, rz=153, fatherId=fPrdFrame[0]}
  [963] = {x=44.636, y=83.455, z=10.804, rx=-171.848, ry=8.891, rz=153, fatherId=fPrdFrame[0]}
  [964] = {x=41.829, y=83.458, z=10.347, rx=-171.856, ry=8.443, rz=153, fatherId=fPrdFrame[0]}
  [965] = {x=39.022, y=83.462, z=9.914, rx=-171.863, ry=7.996, rz=153, fatherId=fPrdFrame[0]}
  [966] = {x=36.216, y=83.465, z=9.504, rx=-171.87, ry=7.549, rz=153, fatherId=fPrdFrame[0]}
  [967] = {x=33.409, y=83.467, z=9.118, rx=-171.877, ry=7.103, rz=153, fatherId=fPrdFrame[0]}
  [968] = {x=30.602, y=83.47, z=8.756, rx=-171.883, ry=6.657, rz=153, fatherId=fPrdFrame[0]}
  [969] = {x=27.795, y=83.473, z=8.418, rx=-171.889, ry=6.211, rz=153, fatherId=fPrdFrame[0]}
  [970] = {x=24.988, y=83.475, z=8.103, rx=-171.894, ry=5.766, rz=153, fatherId=fPrdFrame[0]}
  [971] = {x=22.182, y=83.477, z=7.812, rx=-171.899, ry=5.321, rz=153, fatherId=fPrdFrame[0]}
  [972] = {x=19.375, y=83.479, z=7.545, rx=-171.903, ry=4.877, rz=153, fatherId=fPrdFrame[0]}
  [973] = {x=16.568, y=83.481, z=7.3, rx=-171.907, ry=4.432, rz=153, fatherId=fPrdFrame[0]}
  [974] = {x=13.761, y=83.482, z=7.079, rx=-171.911, ry=3.988, rz=153, fatherId=fPrdFrame[0]}
  [975] = {x=10.954, y=83.484, z=6.882, rx=-171.914, ry=3.545, rz=153, fatherId=fPrdFrame[0]}
  [976] = {x=8.148, y=83.485, z=6.708, rx=-171.917, ry=3.101, rz=153, fatherId=fPrdFrame[0]}
  [977] = {x=5.341, y=83.486, z=6.557, rx=-171.92, ry=2.658, rz=153, fatherId=fPrdFrame[0]}
  [978] = {x=2.534, y=83.487, z=6.429, rx=-171.922, ry=2.215, rz=153, fatherId=fPrdFrame[0]}
  [979] = {x=-0.273, y=83.488, z=6.325, rx=-171.924, ry=1.771, rz=153, fatherId=fPrdFrame[0]}
  [980] = {x=-3.08, y=83.488, z=6.244, rx=-171.925, ry=1.328, rz=153, fatherId=fPrdFrame[0]}
  [981] = {x=-5.886, y=83.489, z=6.186, rx=-171.926, ry=0.886, rz=153, fatherId=fPrdFrame[0]}
  [982] = {x=-8.693, y=83.489, z=6.151, rx=-171.927, ry=0.443, rz=153, fatherId=fPrdFrame[0]}
  [983] = {x=-11.5, y=83.489, z=6.139, rx=-171.927, rz=153, fatherId=fPrdFrame[0]}
  [984] = {x=-14.307, y=83.489, z=6.151, rx=-171.927, ry=-0.443, rz=153, fatherId=fPrdFrame[0]}
  [985] = {x=-17.114, y=83.489, z=6.186, rx=-171.926, ry=-0.886, rz=153, fatherId=fPrdFrame[0]}
  [986] = {x=-19.92, y=83.488, z=6.244, rx=-171.925, ry=-1.328, rz=153, fatherId=fPrdFrame[0]}
  [987] = {x=-22.727, y=83.488, z=6.325, rx=-171.924, ry=-1.771, rz=153, fatherId=fPrdFrame[0]}
  [988] = {x=-25.534, y=83.487, z=6.429, rx=-171.922, ry=-2.215, rz=153, fatherId=fPrdFrame[0]}
  [989] = {x=-28.341, y=83.486, z=6.557, rx=-171.92, ry=-2.658, rz=153, fatherId=fPrdFrame[0]}
  [990] = {x=-31.148, y=83.485, z=6.708, rx=-171.917, ry=-3.101, rz=153, fatherId=fPrdFrame[0]}
  [991] = {x=-33.954, y=83.484, z=6.882, rx=-171.914, ry=-3.545, rz=153, fatherId=fPrdFrame[0]}
  [992] = {x=-36.761, y=83.482, z=7.079, rx=-171.911, ry=-3.988, rz=153, fatherId=fPrdFrame[0]}
  [993] = {x=-39.568, y=83.481, z=7.3, rx=-171.907, ry=-4.432, rz=153, fatherId=fPrdFrame[0]}
  [994] = {x=-42.375, y=83.479, z=7.545, rx=-171.903, ry=-4.877, rz=153, fatherId=fPrdFrame[0]}
  [995] = {x=-45.182, y=83.477, z=7.812, rx=-171.899, ry=-5.321, rz=153, fatherId=fPrdFrame[0]}
  [996] = {x=-47.988, y=83.475, z=8.103, rx=-171.894, ry=-5.766, rz=153, fatherId=fPrdFrame[0]}
  [997] = {x=-50.795, y=83.473, z=8.418, rx=-171.889, ry=-6.211, rz=153, fatherId=fPrdFrame[0]}
  [998] = {x=-53.602, y=83.47, z=8.756, rx=-171.883, ry=-6.657, rz=153, fatherId=fPrdFrame[0]}
  [999] = {x=-56.409, y=83.467, z=9.118, rx=-171.877, ry=-7.103, rz=153, fatherId=fPrdFrame[0]}
string sFileName = "Disk://txt/Toroid_F2_h.txt"
string sMoveMode[1000]
  [0] = "MOVEL"
  [1] = "MOVEL"
  [2] = "MOVEL"
  [3] = "MOVEL"
  [4] = "MOVEL"
  [5] = "MOVEL"
  [6] = "MOVEL"
  [7] = "MOVEL"
  [8] = "MOVEL"
  [9] = "MOVEL"
  [10] = "MOVEL"
  [11] = "MOVEL"
  [12] = "MOVEL"
  [13] = "MOVEL"
  [14] = "MOVEL"
  [15] = "MOVEL"
  [16] = "MOVEL"
  [17] = "MOVEL"
  [18] = "MOVEL"
  [19] = "MOVEL"
  [20] = "MOVEL"
  [21] = "MOVEL"
  [22] = "MOVEL"
  [23] = "MOVEL"
  [24] = "MOVEL"
  [25] = "MOVEL"
  [26] = "MOVEL"
  [27] = "MOVEL"
  [28] = "MOVEL"
  [29] = "MOVEL"
  [30] = "MOVEL"
  [31] = "MOVEL"
  [32] = "MOVEL"
  [33] = "MOVEL"
  [34] = "MOVEL"
  [35] = "MOVEL"
  [36] = "MOVEL"
  [37] = "MOVEL"
  [38] = "MOVEL"
  [39] = "MOVEL"
  [40] = "MOVEL"
  [41] = "MOVEL"
  [42] = "MOVEL"
  [43] = "MOVEL"
  [44] = "MOVEL"
  [45] = "MOVEL"
  [46] = "MOVEL"
  [47] = "MOVEL"
  [48] = "MOVEL"
  [49] = "MOVEL"
  [50] = "MOVEL"
  [51] = "MOVEL"
  [52] = "MOVEL"
  [53] = "MOVEL"
  [54] = "MOVEL"
  [55] = "MOVEL"
  [56] = "MOVEL"
  [57] = "MOVEL"
  [58] = "MOVEL"
  [59] = "MOVEL"
  [60] = "MOVEL"
  [61] = "MOVEL"
  [62] = "MOVEL"
  [63] = "MOVEL"
  [64] = "MOVEL"
  [65] = "MOVEL"
  [66] = "MOVEL"
  [67] = "MOVEL"
  [68] = "MOVEL"
  [69] = "MOVEL"
  [70] = "MOVEL"
  [71] = "MOVEL"
  [72] = "MOVEL"
  [73] = "MOVEL"
  [74] = "MOVEL"
  [75] = "MOVEL"
  [76] = "MOVEL"
  [77] = "MOVEL"
  [78] = "MOVEL"
  [79] = "MOVEL"
  [80] = "MOVEL"
  [81] = "MOVEL"
  [82] = "MOVEL"
  [83] = "MOVEL"
  [84] = "MOVEL"
  [85] = "MOVEL"
  [86] = "MOVEL"
  [87] = "MOVEL"
  [88] = "MOVEL"
  [89] = "MOVEL"
  [90] = "MOVEL"
  [91] = "MOVEL"
  [92] = "MOVEL"
  [93] = "MOVEL"
  [94] = "MOVEL"
  [95] = "MOVEL"
  [96] = "MOVEL"
  [97] = "MOVEL"
  [98] = "MOVEL"
  [99] = "MOVEL"
  [100] = "MOVEL"
  [101] = "MOVEL"
  [102] = "MOVEL"
  [103] = "MOVEL"
  [104] = "MOVEL"
  [105] = "MOVEL"
  [106] = "MOVEL"
  [107] = "MOVEL"
  [108] = "MOVEL"
  [109] = "MOVEL"
  [110] = "MOVEL"
  [111] = "MOVEL"
  [112] = "MOVEL"
  [113] = "MOVEL"
  [114] = "MOVEL"
  [115] = "MOVEL"
  [116] = "MOVEL"
  [117] = "MOVEL"
  [118] = "MOVEL"
  [119] = "MOVEL"
  [120] = "MOVEL"
  [121] = "MOVEL"
  [122] = "MOVEL"
  [123] = "MOVEL"
  [124] = "MOVEL"
  [125] = "MOVEL"
  [126] = "MOVEL"
  [127] = "MOVEL"
  [128] = "MOVEL"
  [129] = "MOVEL"
  [130] = "MOVEL"
  [131] = "MOVEL"
  [132] = "MOVEL"
  [133] = "MOVEL"
  [134] = "MOVEL"
  [135] = "MOVEL"
  [136] = "MOVEL"
  [137] = "MOVEL"
  [138] = "MOVEL"
  [139] = "MOVEL"
  [140] = "MOVEL"
  [141] = "MOVEL"
  [142] = "MOVEL"
  [143] = "MOVEL"
  [144] = "MOVEL"
  [145] = "MOVEL"
  [146] = "MOVEL"
  [147] = "MOVEL"
  [148] = "MOVEL"
  [149] = "MOVEL"
  [150] = "MOVEL"
  [151] = "MOVEL"
  [152] = "MOVEL"
  [153] = "MOVEL"
  [154] = "MOVEL"
  [155] = "MOVEL"
  [156] = "MOVEL"
  [157] = "MOVEL"
  [158] = "MOVEL"
  [159] = "MOVEL"
  [160] = "MOVEL"
  [161] = "MOVEL"
  [162] = "MOVEL"
  [163] = "MOVEL"
  [164] = "MOVEL"
  [165] = "MOVEL"
  [166] = "MOVEL"
  [167] = "MOVEL"
  [168] = "MOVEL"
  [169] = "MOVEL"
  [170] = "MOVEL"
  [171] = "MOVEL"
  [172] = "MOVEL"
  [173] = "MOVEL"
  [174] = "MOVEL"
  [175] = "MOVEL"
  [176] = "MOVEL"
  [177] = "MOVEL"
  [178] = "MOVEL"
  [179] = "MOVEL"
  [180] = "MOVEL"
  [181] = "MOVEL"
  [182] = "MOVEL"
  [183] = "MOVEL"
  [184] = "MOVEL"
  [185] = "MOVEL"
  [186] = "MOVEL"
  [187] = "MOVEL"
  [188] = "MOVEL"
  [189] = "MOVEL"
  [190] = "MOVEL"
  [191] = "MOVEL"
  [192] = "MOVEL"
  [193] = "MOVEL"
  [194] = "MOVEL"
  [195] = "MOVEL"
  [196] = "MOVEL"
  [197] = "MOVEL"
  [198] = "MOVEL"
  [199] = "MOVEL"
  [200] = "MOVEL"
  [201] = "MOVEL"
  [202] = "MOVEL"
  [203] = "MOVEL"
  [204] = "MOVEL"
  [205] = "MOVEL"
  [206] = "MOVEL"
  [207] = "MOVEL"
  [208] = "MOVEL"
  [209] = "MOVEL"
  [210] = "MOVEL"
  [211] = "MOVEL"
  [212] = "MOVEL"
  [213] = "MOVEL"
  [214] = "MOVEL"
  [215] = "MOVEL"
  [216] = "MOVEL"
  [217] = "MOVEL"
  [218] = "MOVEL"
  [219] = "MOVEL"
  [220] = "MOVEL"
  [221] = "MOVEL"
  [222] = "MOVEL"
  [223] = "MOVEL"
  [224] = "MOVEL"
  [225] = "MOVEL"
  [226] = "MOVEL"
  [227] = "MOVEL"
  [228] = "MOVEL"
  [229] = "MOVEL"
  [230] = "MOVEL"
  [231] = "MOVEL"
  [232] = "MOVEL"
  [233] = "MOVEL"
  [234] = "MOVEL"
  [235] = "MOVEL"
  [236] = "MOVEL"
  [237] = "MOVEL"
  [238] = "MOVEL"
  [239] = "MOVEL"
  [240] = "MOVEL"
  [241] = "MOVEL"
  [242] = "MOVEL"
  [243] = "MOVEL"
  [244] = "MOVEL"
  [245] = "MOVEL"
  [246] = "MOVEL"
  [247] = "MOVEL"
  [248] = "MOVEL"
  [249] = "MOVEL"
  [250] = "MOVEL"
  [251] = "MOVEL"
  [252] = "MOVEL"
  [253] = "MOVEL"
  [254] = "MOVEL"
  [255] = "MOVEL"
  [256] = "MOVEL"
  [257] = "MOVEL"
  [258] = "MOVEL"
  [259] = "MOVEL"
  [260] = "MOVEL"
  [261] = "MOVEL"
  [262] = "MOVEL"
  [263] = "MOVEL"
  [264] = "MOVEL"
  [265] = "MOVEL"
  [266] = "MOVEL"
  [267] = "MOVEL"
  [268] = "MOVEL"
  [269] = "MOVEL"
  [270] = "MOVEL"
  [271] = "MOVEL"
  [272] = "MOVEL"
  [273] = "MOVEL"
  [274] = "MOVEL"
  [275] = "MOVEL"
  [276] = "MOVEL"
  [277] = "MOVEL"
  [278] = "MOVEL"
  [279] = "MOVEL"
  [280] = "MOVEL"
  [281] = "MOVEL"
  [282] = "MOVEL"
  [283] = "MOVEL"
  [284] = "MOVEL"
  [285] = "MOVEL"
  [286] = "MOVEL"
  [287] = "MOVEL"
  [288] = "MOVEL"
  [289] = "MOVEL"
  [290] = "MOVEL"
  [291] = "MOVEL"
  [292] = "MOVEL"
  [293] = "MOVEL"
  [294] = "MOVEL"
  [295] = "MOVEL"
  [296] = "MOVEL"
  [297] = "MOVEL"
  [298] = "MOVEL"
  [299] = "MOVEL"
  [300] = "MOVEL"
  [301] = "MOVEL"
  [302] = "MOVEL"
  [303] = "MOVEL"
  [304] = "MOVEL"
  [305] = "MOVEL"
  [306] = "MOVEL"
  [307] = "MOVEL"
  [308] = "MOVEL"
  [309] = "MOVEL"
  [310] = "MOVEL"
  [311] = "MOVEL"
  [312] = "MOVEL"
  [313] = "MOVEL"
  [314] = "MOVEL"
  [315] = "MOVEL"
  [316] = "MOVEL"
  [317] = "MOVEL"
  [318] = "MOVEL"
  [319] = "MOVEL"
  [320] = "MOVEL"
  [321] = "MOVEL"
  [322] = "MOVEL"
  [323] = "MOVEL"
  [324] = "MOVEL"
  [325] = "MOVEL"
  [326] = "MOVEL"
  [327] = "MOVEL"
  [328] = "MOVEL"
  [329] = "MOVEL"
  [330] = "MOVEL"
  [331] = "MOVEL"
  [332] = "MOVEL"
  [333] = "MOVEL"
  [334] = "MOVEL"
  [335] = "MOVEL"
  [336] = "MOVEL"
  [337] = "MOVEL"
  [338] = "MOVEL"
  [339] = "MOVEL"
  [340] = "MOVEL"
  [341] = "MOVEL"
  [342] = "MOVEL"
  [343] = "MOVEL"
  [344] = "MOVEL"
  [345] = "MOVEL"
  [346] = "MOVEL"
  [347] = "MOVEL"
  [348] = "MOVEL"
  [349] = "MOVEL"
  [350] = "MOVEL"
  [351] = "MOVEL"
  [352] = "MOVEL"
  [353] = "MOVEL"
  [354] = "MOVEL"
  [355] = "MOVEL"
  [356] = "MOVEL"
  [357] = "MOVEL"
  [358] = "MOVEL"
  [359] = "MOVEL"
  [360] = "MOVEL"
  [361] = "MOVEL"
  [362] = "MOVEL"
  [363] = "MOVEL"
  [364] = "MOVEL"
  [365] = "MOVEL"
  [366] = "MOVEL"
  [367] = "MOVEL"
  [368] = "MOVEL"
  [369] = "MOVEL"
  [370] = "MOVEL"
  [371] = "MOVEL"
  [372] = "MOVEL"
  [373] = "MOVEL"
  [374] = "MOVEL"
  [375] = "MOVEL"
  [376] = "MOVEL"
  [377] = "MOVEL"
  [378] = "MOVEL"
  [379] = "MOVEL"
  [380] = "MOVEL"
  [381] = "MOVEL"
  [382] = "MOVEL"
  [383] = "MOVEL"
  [384] = "MOVEL"
  [385] = "MOVEL"
  [386] = "MOVEL"
  [387] = "MOVEL"
  [388] = "MOVEL"
  [389] = "MOVEL"
  [390] = "MOVEL"
  [391] = "MOVEL"
  [392] = "MOVEL"
  [393] = "MOVEL"
  [394] = "MOVEL"
  [395] = "MOVEL"
  [396] = "MOVEL"
  [397] = "MOVEL"
  [398] = "MOVEL"
  [399] = "MOVEL"
  [400] = "MOVEL"
  [401] = "MOVEL"
  [402] = "MOVEL"
  [403] = "MOVEL"
  [404] = "MOVEL"
  [405] = "MOVEL"
  [406] = "MOVEL"
  [407] = "MOVEL"
  [408] = "MOVEL"
  [409] = "MOVEL"
  [410] = "MOVEL"
  [411] = "MOVEL"
  [412] = "MOVEL"
  [413] = "MOVEL"
  [414] = "MOVEL"
  [415] = "MOVEL"
  [416] = "MOVEL"
  [417] = "MOVEL"
  [418] = "MOVEL"
  [419] = "MOVEL"
  [420] = "MOVEL"
  [421] = "MOVEL"
  [422] = "MOVEL"
  [423] = "MOVEL"
  [424] = "MOVEL"
  [425] = "MOVEL"
  [426] = "MOVEL"
  [427] = "MOVEL"
  [428] = "MOVEL"
  [429] = "MOVEL"
  [430] = "MOVEL"
  [431] = "MOVEL"
  [432] = "MOVEL"
  [433] = "MOVEL"
  [434] = "MOVEL"
  [435] = "MOVEL"
  [436] = "MOVEL"
  [437] = "MOVEL"
  [438] = "MOVEL"
  [439] = "MOVEL"
  [440] = "MOVEL"
  [441] = "MOVEL"
  [442] = "MOVEL"
  [443] = "MOVEL"
  [444] = "MOVEL"
  [445] = "MOVEL"
  [446] = "MOVEL"
  [447] = "MOVEL"
  [448] = "MOVEL"
  [449] = "MOVEL"
  [450] = "MOVEL"
  [451] = "MOVEL"
  [452] = "MOVEL"
  [453] = "MOVEL"
  [454] = "MOVEL"
  [455] = "MOVEL"
  [456] = "MOVEL"
  [457] = "MOVEL"
  [458] = "MOVEL"
  [459] = "MOVEL"
  [460] = "MOVEL"
  [461] = "MOVEL"
  [462] = "MOVEL"
  [463] = "MOVEL"
  [464] = "MOVEL"
  [465] = "MOVEL"
  [466] = "MOVEL"
  [467] = "MOVEL"
  [468] = "MOVEL"
  [469] = "MOVEL"
  [470] = "MOVEL"
  [471] = "MOVEL"
  [472] = "MOVEL"
  [473] = "MOVEL"
  [474] = "MOVEL"
  [475] = "MOVEL"
  [476] = "MOVEL"
  [477] = "MOVEL"
  [478] = "MOVEL"
  [479] = "MOVEL"
  [480] = "MOVEL"
  [481] = "MOVEL"
  [482] = "MOVEL"
  [483] = "MOVEL"
  [484] = "MOVEL"
  [485] = "MOVEL"
  [486] = "MOVEL"
  [487] = "MOVEL"
  [488] = "MOVEL"
  [489] = "MOVEL"
  [490] = "MOVEL"
  [491] = "MOVEL"
  [492] = "MOVEL"
  [493] = "MOVEL"
  [494] = "MOVEL"
  [495] = "MOVEL"
  [496] = "MOVEL"
  [497] = "MOVEL"
  [498] = "MOVEJ"
  [499] = "MOVEL"
  [500] = "MOVEL"
  [501] = "MOVEL"
  [502] = "MOVEL"
  [503] = "MOVEL"
  [504] = "MOVEL"
  [505] = "MOVEL"
  [506] = "MOVEL"
  [507] = "MOVEL"
  [508] = "MOVEL"
  [509] = "MOVEL"
  [510] = "MOVEL"
  [511] = "MOVEL"
  [512] = "MOVEL"
  [513] = "MOVEL"
  [514] = "MOVEL"
  [515] = "MOVEL"
  [516] = "MOVEL"
  [517] = "MOVEL"
  [518] = "MOVEL"
  [519] = "MOVEL"
  [520] = "MOVEL"
  [521] = "MOVEL"
  [522] = "MOVEL"
  [523] = "MOVEL"
  [524] = "MOVEL"
  [525] = "MOVEL"
  [526] = "MOVEL"
  [527] = "MOVEL"
  [528] = "MOVEL"
  [529] = "MOVEL"
  [530] = "MOVEL"
  [531] = "MOVEL"
  [532] = "MOVEL"
  [533] = "MOVEL"
  [534] = "MOVEL"
  [535] = "MOVEL"
  [536] = "MOVEL"
  [537] = "MOVEL"
  [538] = "MOVEL"
  [539] = "MOVEL"
  [540] = "MOVEL"
  [541] = "MOVEL"
  [542] = "MOVEL"
  [543] = "MOVEL"
  [544] = "MOVEL"
  [545] = "MOVEL"
  [546] = "MOVEL"
  [547] = "MOVEL"
  [548] = "MOVEL"
  [549] = "MOVEL"
  [550] = "MOVEL"
  [551] = "MOVEL"
  [552] = "MOVEL"
  [553] = "MOVEL"
  [554] = "MOVEL"
  [555] = "MOVEL"
  [556] = "MOVEL"
  [557] = "MOVEL"
  [558] = "MOVEL"
  [559] = "MOVEL"
  [560] = "MOVEL"
  [561] = "MOVEL"
  [562] = "MOVEL"
  [563] = "MOVEL"
  [564] = "MOVEL"
  [565] = "MOVEL"
  [566] = "MOVEL"
  [567] = "MOVEL"
  [568] = "MOVEL"
  [569] = "MOVEL"
  [570] = "MOVEL"
  [571] = "MOVEL"
  [572] = "MOVEL"
  [573] = "MOVEL"
  [574] = "MOVEL"
  [575] = "MOVEL"
  [576] = "MOVEL"
  [577] = "MOVEL"
  [578] = "MOVEL"
  [579] = "MOVEL"
  [580] = "MOVEL"
  [581] = "MOVEL"
  [582] = "MOVEL"
  [583] = "MOVEL"
  [584] = "MOVEL"
  [585] = "MOVEL"
  [586] = "MOVEL"
  [587] = "MOVEL"
  [588] = "MOVEL"
  [589] = "MOVEL"
  [590] = "MOVEL"
  [591] = "MOVEL"
  [592] = "MOVEL"
  [593] = "MOVEL"
  [594] = "MOVEL"
  [595] = "MOVEL"
  [596] = "MOVEL"
  [597] = "MOVEL"
  [598] = "MOVEL"
  [599] = "MOVEL"
  [600] = "MOVEL"
  [601] = "MOVEL"
  [602] = "MOVEL"
  [603] = "MOVEL"
  [604] = "MOVEL"
  [605] = "MOVEL"
  [606] = "MOVEL"
  [607] = "MOVEL"
  [608] = "MOVEL"
  [609] = "MOVEL"
  [610] = "MOVEL"
  [611] = "MOVEL"
  [612] = "MOVEL"
  [613] = "MOVEL"
  [614] = "MOVEL"
  [615] = "MOVEL"
  [616] = "MOVEL"
  [617] = "MOVEL"
  [618] = "MOVEL"
  [619] = "MOVEL"
  [620] = "MOVEL"
  [621] = "MOVEL"
  [622] = "MOVEL"
  [623] = "MOVEL"
  [624] = "MOVEL"
  [625] = "MOVEL"
  [626] = "MOVEL"
  [627] = "MOVEL"
  [628] = "MOVEL"
  [629] = "MOVEL"
  [630] = "MOVEL"
  [631] = "MOVEL"
  [632] = "MOVEL"
  [633] = "MOVEL"
  [634] = "MOVEL"
  [635] = "MOVEL"
  [636] = "MOVEL"
  [637] = "MOVEL"
  [638] = "MOVEL"
  [639] = "MOVEL"
  [640] = "MOVEL"
  [641] = "MOVEL"
  [642] = "MOVEL"
  [643] = "MOVEL"
  [644] = "MOVEL"
  [645] = "MOVEL"
  [646] = "MOVEL"
  [647] = "MOVEL"
  [648] = "MOVEL"
  [649] = "MOVEL"
  [650] = "MOVEL"
  [651] = "MOVEL"
  [652] = "MOVEL"
  [653] = "MOVEL"
  [654] = "MOVEL"
  [655] = "MOVEL"
  [656] = "MOVEL"
  [657] = "MOVEL"
  [658] = "MOVEL"
  [659] = "MOVEL"
  [660] = "MOVEL"
  [661] = "MOVEL"
  [662] = "MOVEL"
  [663] = "MOVEL"
  [664] = "MOVEL"
  [665] = "MOVEL"
  [666] = "MOVEL"
  [667] = "MOVEL"
  [668] = "MOVEL"
  [669] = "MOVEL"
  [670] = "MOVEL"
  [671] = "MOVEL"
  [672] = "MOVEL"
  [673] = "MOVEL"
  [674] = "MOVEL"
  [675] = "MOVEL"
  [676] = "MOVEL"
  [677] = "MOVEL"
  [678] = "MOVEL"
  [679] = "MOVEL"
  [680] = "MOVEL"
  [681] = "MOVEL"
  [682] = "MOVEL"
  [683] = "MOVEL"
  [684] = "MOVEL"
  [685] = "MOVEL"
  [686] = "MOVEL"
  [687] = "MOVEL"
  [688] = "MOVEL"
  [689] = "MOVEL"
  [690] = "MOVEL"
  [691] = "MOVEL"
  [692] = "MOVEL"
  [693] = "MOVEL"
  [694] = "MOVEL"
  [695] = "MOVEL"
  [696] = "MOVEL"
  [697] = "MOVEL"
  [698] = "MOVEL"
  [699] = "MOVEL"
  [700] = "MOVEL"
  [701] = "MOVEL"
  [702] = "MOVEL"
  [703] = "MOVEL"
  [704] = "MOVEL"
  [705] = "MOVEL"
  [706] = "MOVEL"
  [707] = "MOVEL"
  [708] = "MOVEL"
  [709] = "MOVEL"
  [710] = "MOVEL"
  [711] = "MOVEL"
  [712] = "MOVEL"
  [713] = "MOVEL"
  [714] = "MOVEL"
  [715] = "MOVEL"
  [716] = "MOVEL"
  [717] = "MOVEL"
  [718] = "MOVEL"
  [719] = "MOVEL"
  [720] = "MOVEL"
  [721] = "MOVEL"
  [722] = "MOVEL"
  [723] = "MOVEL"
  [724] = "MOVEL"
  [725] = "MOVEL"
  [726] = "MOVEL"
  [727] = "MOVEL"
  [728] = "MOVEL"
  [729] = "MOVEL"
  [730] = "MOVEL"
  [731] = "MOVEL"
  [732] = "MOVEL"
  [733] = "MOVEL"
  [734] = "MOVEL"
  [735] = "MOVEL"
  [736] = "MOVEL"
  [737] = "MOVEL"
  [738] = "MOVEL"
  [739] = "MOVEL"
  [740] = "MOVEL"
  [741] = "MOVEL"
  [742] = "MOVEL"
  [743] = "MOVEL"
  [744] = "MOVEL"
  [745] = "MOVEL"
  [746] = "MOVEL"
  [747] = "MOVEL"
  [748] = "MOVEL"
  [749] = "MOVEL"
  [750] = "MOVEL"
  [751] = "MOVEL"
  [752] = "MOVEL"
  [753] = "MOVEL"
  [754] = "MOVEL"
  [755] = "MOVEL"
  [756] = "MOVEL"
  [757] = "MOVEL"
  [758] = "MOVEL"
  [759] = "MOVEL"
  [760] = "MOVEL"
  [761] = "MOVEL"
  [762] = "MOVEL"
  [763] = "MOVEL"
  [764] = "MOVEL"
  [765] = "MOVEL"
  [766] = "MOVEL"
  [767] = "MOVEL"
  [768] = "MOVEL"
  [769] = "MOVEL"
  [770] = "MOVEL"
  [771] = "MOVEL"
  [772] = "MOVEL"
  [773] = "MOVEL"
  [774] = "MOVEL"
  [775] = "MOVEL"
  [776] = "MOVEL"
  [777] = "MOVEL"
  [778] = "MOVEL"
  [779] = "MOVEL"
  [780] = "MOVEL"
  [781] = "MOVEL"
  [782] = "MOVEL"
  [783] = "MOVEL"
  [784] = "MOVEL"
  [785] = "MOVEL"
  [786] = "MOVEL"
  [787] = "MOVEL"
  [788] = "MOVEL"
  [789] = "MOVEL"
  [790] = "MOVEL"
  [791] = "MOVEL"
  [792] = "MOVEL"
  [793] = "MOVEL"
  [794] = "MOVEL"
  [795] = "MOVEL"
  [796] = "MOVEL"
  [797] = "MOVEL"
  [798] = "MOVEL"
  [799] = "MOVEL"
  [800] = "MOVEL"
  [801] = "MOVEL"
  [802] = "MOVEL"
  [803] = "MOVEL"
  [804] = "MOVEL"
  [805] = "MOVEL"
  [806] = "MOVEL"
  [807] = "MOVEL"
  [808] = "MOVEL"
  [809] = "MOVEL"
  [810] = "MOVEL"
  [811] = "MOVEL"
  [812] = "MOVEL"
  [813] = "MOVEL"
  [814] = "MOVEL"
  [815] = "MOVEL"
  [816] = "MOVEL"
  [817] = "MOVEL"
  [818] = "MOVEL"
  [819] = "MOVEL"
  [820] = "MOVEL"
  [821] = "MOVEL"
  [822] = "MOVEL"
  [823] = "MOVEL"
  [824] = "MOVEL"
  [825] = "MOVEL"
  [826] = "MOVEL"
  [827] = "MOVEL"
  [828] = "MOVEL"
  [829] = "MOVEL"
  [830] = "MOVEL"
  [831] = "MOVEL"
  [832] = "MOVEL"
  [833] = "MOVEL"
  [834] = "MOVEL"
  [835] = "MOVEL"
  [836] = "MOVEL"
  [837] = "MOVEL"
  [838] = "MOVEL"
  [839] = "MOVEL"
  [840] = "MOVEL"
  [841] = "MOVEL"
  [842] = "MOVEL"
  [843] = "MOVEL"
  [844] = "MOVEL"
  [845] = "MOVEL"
  [846] = "MOVEL"
  [847] = "MOVEL"
  [848] = "MOVEL"
  [849] = "MOVEL"
  [850] = "MOVEL"
  [851] = "MOVEL"
  [852] = "MOVEL"
  [853] = "MOVEL"
  [854] = "MOVEL"
  [855] = "MOVEL"
  [856] = "MOVEL"
  [857] = "MOVEL"
  [858] = "MOVEL"
  [859] = "MOVEL"
  [860] = "MOVEL"
  [861] = "MOVEL"
  [862] = "MOVEL"
  [863] = "MOVEL"
  [864] = "MOVEL"
  [865] = "MOVEL"
  [866] = "MOVEL"
  [867] = "MOVEL"
  [868] = "MOVEL"
  [869] = "MOVEL"
  [870] = "MOVEL"
  [871] = "MOVEL"
  [872] = "MOVEL"
  [873] = "MOVEL"
  [874] = "MOVEL"
  [875] = "MOVEL"
  [876] = "MOVEL"
  [877] = "MOVEL"
  [878] = "MOVEL"
  [879] = "MOVEL"
  [880] = "MOVEL"
  [881] = "MOVEL"
  [882] = "MOVEL"
  [883] = "MOVEL"
  [884] = "MOVEL"
  [885] = "MOVEL"
  [886] = "MOVEL"
  [887] = "MOVEL"
  [888] = "MOVEL"
  [889] = "MOVEL"
  [890] = "MOVEL"
  [891] = "MOVEL"
  [892] = "MOVEL"
  [893] = "MOVEL"
  [894] = "MOVEL"
  [895] = "MOVEL"
  [896] = "MOVEL"
  [897] = "MOVEL"
  [898] = "MOVEL"
  [899] = "MOVEL"
  [900] = "MOVEL"
  [901] = "MOVEL"
  [902] = "MOVEL"
  [903] = "MOVEL"
  [904] = "MOVEL"
  [905] = "MOVEL"
  [906] = "MOVEL"
  [907] = "MOVEL"
  [908] = "MOVEL"
  [909] = "MOVEL"
  [910] = "MOVEL"
  [911] = "MOVEL"
  [912] = "MOVEL"
  [913] = "MOVEL"
  [914] = "MOVEL"
  [915] = "MOVEL"
  [916] = "MOVEL"
  [917] = "MOVEL"
  [918] = "MOVEL"
  [919] = "MOVEL"
  [920] = "MOVEL"
  [921] = "MOVEL"
  [922] = "MOVEL"
  [923] = "MOVEL"
  [924] = "MOVEL"
  [925] = "MOVEL"
  [926] = "MOVEL"
  [927] = "MOVEL"
  [928] = "MOVEL"
  [929] = "MOVEL"
  [930] = "MOVEL"
  [931] = "MOVEL"
  [932] = "MOVEL"
  [933] = "MOVEL"
  [934] = "MOVEL"
  [935] = "MOVEL"
  [936] = "MOVEL"
  [937] = "MOVEL"
  [938] = "MOVEL"
  [939] = "MOVEL"
  [940] = "MOVEL"
  [941] = "MOVEL"
  [942] = "MOVEL"
  [943] = "MOVEL"
  [944] = "MOVEL"
  [945] = "MOVEL"
  [946] = "MOVEL"
  [947] = "MOVEL"
  [948] = "MOVEL"
  [949] = "MOVEL"
  [950] = "MOVEL"
  [951] = "MOVEL"
  [952] = "MOVEL"
  [953] = "MOVEL"
  [954] = "MOVEL"
  [955] = "MOVEL"
  [956] = "MOVEL"
  [957] = "MOVEL"
  [958] = "MOVEL"
  [959] = "MOVEL"
  [960] = "MOVEL"
  [961] = "MOVEL"
  [962] = "MOVEL"
  [963] = "MOVEL"
  [964] = "MOVEL"
  [965] = "MOVEL"
  [966] = "MOVEL"
  [967] = "MOVEL"
  [968] = "MOVEL"
  [969] = "MOVEL"
  [970] = "MOVEL"
  [971] = "MOVEL"
  [972] = "MOVEL"
  [973] = "MOVEL"
  [974] = "MOVEL"
  [975] = "MOVEL"
  [976] = "MOVEL"
  [977] = "MOVEL"
  [978] = "MOVEL"
  [979] = "MOVEL"
  [980] = "MOVEL"
  [981] = "MOVEL"
  [982] = "MOVEL"
  [983] = "MOVEL"
  [984] = "MOVEL"
  [985] = "MOVEL"
  [986] = "MOVEL"
  [987] = "MOVEL"
  [988] = "MOVEL"
  [989] = "MOVEL"
  [990] = "MOVEL"
  [991] = "MOVEL"
  [992] = "MOVEL"
  [993] = "MOVEL"
  [994] = "MOVEL"
  [995] = "MOVEL"
  [996] = "MOVEL"
  [997] = "MOVEL"
  [998] = "MOVEL"
  [999] = "MOVEL"
string sPrdID = "Toroid_F2_h"
string sSpeedDate = "  0   "
public tool tPrdTool = {x=350.215, y=-0.767, z=232.539, rx=-89.841, ry=89.729, rz=89.842, fatherId=flange[0], ioLink=valve1}
trsf trPrdFrmOffset
